    movel([0.119782, -1.382241, -2.558201, -0.771947, 1.570796, 1.690578],accel_mss,speed_ms,0,blend_radius_m)
    speed_ms = 1.000
    movel([0.119782, -1.357452, -2.545969, -0.808968, 1.570796, 1.690578],accel_mss,speed_ms,0,blend_radius_m)
    movel([0.118569, -1.359477, -2.544576, -0.808336, 1.570796, 1.689365],accel_mss,speed_ms,0,blend_radius_m)
    movel([0.118569, -1.384229, -2.556783, -0.771377, 1.570796, 1.689365],accel_mss,speed_ms,0,blend_radius_m)
    speed_ms = 0.003
    movel([0.118569, -1.393867, -2.561225, -0.757297, 1.570796, 1.689365],accel_mss,speed_ms,0,blend_radius_m)
    speed_ms = 0.007
    movel([0.118728, -1.394054, -2.561089, -0.757246, 1.570796, 1.689524],accel_mss,speed_ms,0,blend_radius_m)
    movel([0.118593, -1.394865, -2.560501, -0.757024, 1.570796, 1.689390],accel_mss,speed_ms,0,blend_radius_m)
    movel([0.118424, -1.395809, -2.559814, -0.756766, 1.570796, 1.689220],accel_mss,speed_ms,0,blend_radius_m)
    movel([0.118206, -1.396901, -2.559018, -0.756470, 1.570796, 1.689002],accel_mss,speed_ms,0,blend_radius_m)
    movel([0.117896, -1.398373, -2.557942, -0.756074, 1.570796, 1.688693],accel_mss,speed_ms,0,blend_radius_m)
    movel([0.117699, -1.399201, -2.557336, -0.755852, 1.570796, 1.688495],accel_mss,speed_ms,0,blend_radius_m)
    movel([0.117545, -1.399729, -2.556948, -0.755712, 1.570796, 1.688341],accel_mss,speed_ms,0,blend_radius_m)
    movel([0.117303, -1.400036, -2.556723, -0.755630, 1.570796, 1.688099],accel_mss,speed_ms,0,blend_radius_m)
    movel([0.117055, -1.400079, -2.556692, -0.755619, 1.570796, 1.687851],accel_mss,speed_ms,0,blend_radius_m)
    movel([0.117023, -1.399429, -2.557168, -0.755792, 1.570796, 1.687819],accel_mss,speed_ms,0,blend_radius_m)
    movel([0.117111, -1.398603, -2.557774, -0.756012, 1.570796, 1.687907],accel_mss,speed_ms,0,blend_radius_m)
    movel([0.117305, -1.397157, -2.558831, -0.756401, 1.570796, 1.688101],accel_mss,speed_ms,0,blend_radius_m)
    movel([0.117464, -1.396051, -2.559637, -0.756700, 1.570796, 1.688261],accel_mss,speed_ms,0,blend_radius_m)
    movel([0.117616, -1.395092, -2.560336, -0.756962, 1.570796, 1.688412],accel_mss,speed_ms,0,blend_radius_m)
    movel([0.117758, -1.394259, -2.560940, -0.757189, 1.570796, 1.688554],accel_mss,speed_ms,0,blend_radius_m)
    movel([0.117985, -1.394001, -2.561128, -0.757260, 1.570796, 1.688781],accel_mss,speed_ms,0,blend_radius_m)
    movel([0.118280, -1.393900, -2.561201, -0.757288, 1.570796, 1.689077],accel_mss,speed_ms,0,blend_radius_m)
    movel([0.118569, -1.393867, -2.561225, -0.757297, 1.570796, 1.689365],accel_mss,speed_ms,0,blend_radius_m)
    speed_ms = 0.003
    movel([0.118569, -1.397123, -2.562689, -0.752577, 1.570796, 1.689365],accel_mss,speed_ms,0,blend_radius_m)
    speed_ms = 0.007
    movel([0.118728, -1.397310, -2.562553, -0.752526, 1.570796, 1.689524],accel_mss,speed_ms,0,blend_radius_m)
    movel([0.118593, -1.398118, -2.561963, -0.752308, 1.570796, 1.689390],accel_mss,speed_ms,0,blend_radius_m)
    movel([0.118424, -1.399059, -2.561275, -0.752055, 1.570796, 1.689220],accel_mss,speed_ms,0,blend_radius_m)
    movel([0.118206, -1.400148, -2.560477, -0.751764, 1.570796, 1.689002],accel_mss,speed_ms,0,blend_radius_m)
    movel([0.117896, -1.401617, -2.559399, -0.751374, 1.570796, 1.688693],accel_mss,speed_ms,0,blend_radius_m)
    movel([0.117699, -1.402442, -2.558791, -0.751156, 1.570796, 1.688495],accel_mss,speed_ms,0,blend_radius_m)
    movel([0.117545, -1.402968, -2.558403, -0.751018, 1.570796, 1.688341],accel_mss,speed_ms,0,blend_radius_m)
    movel([0.117303, -1.403274, -2.558177, -0.750937, 1.570796, 1.688099],accel_mss,speed_ms,0,blend_radius_m)
    movel([0.117055, -1.403317, -2.558145, -0.750926, 1.570796, 1.687851],accel_mss,speed_ms,0,blend_radius_m)
    movel([0.117023, -1.402670, -2.558623, -0.751096, 1.570796, 1.687819],accel_mss,speed_ms,0,blend_radius_m)
    movel([0.117111, -1.401846, -2.559230, -0.751313, 1.570796, 1.687907],accel_mss,speed_ms,0,blend_radius_m)
    movel([0.117305, -1.400404, -2.560290, -0.751696, 1.570796, 1.688101],accel_mss,speed_ms,0,blend_radius_m)
    movel([0.117464, -1.399301, -2.561098, -0.751990, 1.570796, 1.688261],accel_mss,speed_ms,0,blend_radius_m)
    movel([0.117616, -1.398344, -2.561798, -0.752247, 1.570796, 1.688412],accel_mss,speed_ms,0,blend_radius_m)
    movel([0.117758, -1.397514, -2.562404, -0.752471, 1.570796, 1.688554],accel_mss,speed_ms,0,blend_radius_m)
    movel([0.117985, -1.397256, -2.562592, -0.752541, 1.570796, 1.688781],accel_mss,speed_ms,0,blend_radius_m)
    movel([0.118280, -1.397156, -2.562665, -0.752568, 1.570796, 1.689077],accel_mss,speed_ms,0,blend_radius_m)
    movel([0.118569, -1.397123, -2.562689, -0.752577, 1.570796, 1.689365],accel_mss,speed_ms,0,blend_radius_m)
    speed_ms = 0.003
    movel([0.118569, -1.384229, -2.556783, -0.771377, 1.570796, 1.689365],accel_mss,speed_ms,0,blend_radius_m)
    speed_ms = 1.000
    movel([0.118569, -1.359477, -2.544576, -0.808336, 1.570796, 1.689365],accel_mss,speed_ms,0,blend_radius_m)
    movel([0.118605, -1.358852, -2.545007, -0.808530, 1.570796, 1.689401],accel_mss,speed_ms,0,blend_radius_m)
    movel([0.118605, -1.383615, -2.557221, -0.771552, 1.570796, 1.689401],accel_mss,speed_ms,0,blend_radius_m)
    speed_ms = 0.003
    movel([0.118605, -1.393258, -2.561667, -0.757465, 1.570796, 1.689401],accel_mss,speed_ms,0,blend_radius_m)
    speed_ms = 0.007
    movel([0.118234, -1.393393, -2.561569, -0.757427, 1.570796, 1.689030],accel_mss,speed_ms,0,blend_radius_m)
    movel([0.117908, -1.393450, -2.561527, -0.757412, 1.570796, 1.688705],accel_mss,speed_ms,0,blend_radius_m)
    movel([0.117689, -1.393424, -2.561546, -0.757419, 1.570796, 1.688485],accel_mss,speed_ms,0,blend_radius_m)
    movel([0.117549, -1.393131, -2.561759, -0.757500, 1.570796, 1.688345],accel_mss,speed_ms,0,blend_radius_m)
    movel([0.117522, -1.392806, -2.561994, -0.757589, 1.570796, 1.688318],accel_mss,speed_ms,0,blend_radius_m)
    movel([0.117346, -1.392422, -2.562271, -0.757695, 1.570796, 1.688142],accel_mss,speed_ms,0,blend_radius_m)
    movel([0.117088, -1.392080, -2.562518, -0.757790, 1.570796, 1.687885],accel_mss,speed_ms,0,blend_radius_m)
    movel([0.116802, -1.391882, -2.562661, -0.757845, 1.570796, 1.687598],accel_mss,speed_ms,0,blend_radius_m)
    movel([0.116439, -1.391787, -2.562731, -0.757872, 1.570796, 1.687236],accel_mss,speed_ms,0,blend_radius_m)
    movel([0.116040, -1.391804, -2.562718, -0.757867, 1.570796, 1.686837],accel_mss,speed_ms,0,blend_radius_m)
    movel([0.115619, -1.391935, -2.562624, -0.757831, 1.570796, 1.686415],accel_mss,speed_ms,0,blend_radius_m)
    movel([0.115183, -1.392176, -2.562449, -0.757764, 1.570796, 1.685979],accel_mss,speed_ms,0,blend_radius_m)
    movel([0.114712, -1.392597, -2.562145, -0.757647, 1.570796, 1.685508],accel_mss,speed_ms,0,blend_radius_m)
    movel([0.114471, -1.393051, -2.561816, -0.757522, 1.570796, 1.685267],accel_mss,speed_ms,0,blend_radius_m)
    movel([0.114501, -1.393491, -2.561498, -0.757401, 1.570796, 1.685297],accel_mss,speed_ms,0,blend_radius_m)
    movel([0.114790, -1.393868, -2.561224, -0.757297, 1.570796, 1.685586],accel_mss,speed_ms,0,blend_radius_m)
    movel([0.115093, -1.394046, -2.561095, -0.757248, 1.570796, 1.685889],accel_mss,speed_ms,0,blend_radius_m)
    movel([0.115465, -1.394151, -2.561019, -0.757219, 1.570796, 1.686262],accel_mss,speed_ms,0,blend_radius_m)
    movel([0.115948, -1.394188, -2.560992, -0.757209, 1.570796, 1.686745],accel_mss,speed_ms,0,blend_radius_m)
    movel([0.116596, -1.394166, -2.561008, -0.757215, 1.570796, 1.687392],accel_mss,speed_ms,0,blend_radius_m)
    movel([0.116840, -1.394198, -2.560985, -0.757206, 1.570796, 1.687637],accel_mss,speed_ms,0,blend_radius_m)
    movel([0.117037, -1.394702, -2.560619, -0.757068, 1.570796, 1.687833],accel_mss,speed_ms,0,blend_radius_m)
    movel([0.116741, -1.397152, -2.558834, -0.756402, 1.570796, 1.687538],accel_mss,speed_ms,0,blend_radius_m)
    movel([0.116430, -1.399585, -2.557054, -0.755750, 1.570796, 1.687226],accel_mss,speed_ms,0,blend_radius_m)
    movel([0.116267, -1.400079, -2.556692, -0.755619, 1.570796, 1.687063],accel_mss,speed_ms,0,blend_radius_m)
    movel([0.116071, -1.400343, -2.556497, -0.755549, 1.570796, 1.686867],accel_mss,speed_ms,0,blend_radius_m)
    movel([0.115806, -1.400476, -2.556399, -0.755513, 1.570796, 1.686603],accel_mss,speed_ms,0,blend_radius_m)
    movel([0.115532, -1.400483, -2.556394, -0.755511, 1.570796, 1.686329],accel_mss,speed_ms,0,blend_radius_m)
    movel([0.115371, -1.400354, -2.556490, -0.755546, 1.570796, 1.686167],accel_mss,speed_ms,0,blend_radius_m)
    movel([0.115306, -1.400032, -2.556726, -0.755631, 1.570796, 1.686102],accel_mss,speed_ms,0,blend_radius_m)
    movel([0.115324, -1.399384, -2.557202, -0.755804, 1.570796, 1.686120],accel_mss,speed_ms,0,blend_radius_m)
    movel([0.115335, -1.399019, -2.557469, -0.755901, 1.570796, 1.686131],accel_mss,speed_ms,0,blend_radius_m)
    movel([0.115328, -1.398702, -2.557701, -0.755986, 1.570796, 1.686124],accel_mss,speed_ms,0,blend_radius_m)
    movel([0.115303, -1.398449, -2.557887, -0.756054, 1.570796, 1.686099],accel_mss,speed_ms,0,blend_radius_m)
    movel([0.114943, -1.398374, -2.557941, -0.756074, 1.570796, 1.685739],accel_mss,speed_ms,0,blend_radius_m)
    movel([0.114662, -1.398389, -2.557930, -0.756070, 1.570796, 1.685459],accel_mss,speed_ms,0,blend_radius_m)
    movel([0.114357, -1.398417, -2.557910, -0.756062, 1.570796, 1.685153],accel_mss,speed_ms,0,blend_radius_m)
    movel([0.112719, -1.398331, -2.557973, -0.756085, 1.570796, 1.683515],accel_mss,speed_ms,0,blend_radius_m)
    movel([0.111315, -1.397718, -2.558421, -0.756250, 1.570796, 1.682112],accel_mss,speed_ms,0,blend_radius_m)
    movel([0.110329, -1.396670, -2.559187, -0.756533, 1.570796, 1.681125],accel_mss,speed_ms,0,blend_radius_m)
    movel([0.109898, -1.395312, -2.560175, -0.756901, 1.570796, 1.680695],accel_mss,speed_ms,0,blend_radius_m)
    movel([0.110008, -1.393931, -2.561179, -0.757279, 1.570796, 1.680804],accel_mss,speed_ms,0,blend_radius_m)
    movel([0.110561, -1.392374, -2.562306, -0.757709, 1.570796, 1.681357],accel_mss,speed_ms,0,blend_radius_m)
    movel([0.111504, -1.390778, -2.563459, -0.758153, 1.570796, 1.682300],accel_mss,speed_ms,0,blend_radius_m)
    movel([0.112755, -1.389292, -2.564528, -0.758569, 1.570796, 1.683551],accel_mss,speed_ms,0,blend_radius_m)
    movel([0.113901, -1.388249, -2.565277, -0.758863, 1.570796, 1.684697],accel_mss,speed_ms,0,blend_radius_m)
    movel([0.115113, -1.387370, -2.565906, -0.759112, 1.570796, 1.685909],accel_mss,speed_ms,0,blend_radius_m)
    movel([0.116414, -1.386641, -2.566428, -0.759320, 1.570796, 1.687210],accel_mss,speed_ms,0,blend_radius_m)
    movel([0.117832, -1.386048, -2.566851, -0.759489, 1.570796, 1.688629],accel_mss,speed_ms,0,blend_radius_m)
    movel([0.119207, -1.385643, -2.567141, -0.759605, 1.570796, 1.690004],accel_mss,speed_ms,0,blend_radius_m)
    movel([0.120533, -1.385423, -2.567298, -0.759669, 1.570796, 1.691329],accel_mss,speed_ms,0,blend_radius_m)
    movel([0.121802, -1.385387, -2.567323, -0.759679, 1.570796, 1.692598],accel_mss,speed_ms,0,blend_radius_m)
    movel([0.123004, -1.385538, -2.567216, -0.759636, 1.570796, 1.693800],accel_mss,speed_ms,0,blend_radius_m)
    movel([0.124432, -1.386000, -2.566886, -0.759503, 1.570796, 1.695228],accel_mss,speed_ms,0,blend_radius_m)
    movel([0.125530, -1.386717, -2.566374, -0.759299, 1.570796, 1.696327],accel_mss,speed_ms,0,blend_radius_m)
    movel([0.126289, -1.387678, -2.565686, -0.759025, 1.570796, 1.697085],accel_mss,speed_ms,0,blend_radius_m)
    movel([0.126698, -1.388871, -2.564830, -0.758688, 1.570796, 1.697494],accel_mss,speed_ms,0,blend_radius_m)
    movel([0.126745, -1.389618, -2.564293, -0.758477, 1.570796, 1.697542],accel_mss,speed_ms,0,blend_radius_m)
    movel([0.126649, -1.390509, -2.563652, -0.758228, 1.570796, 1.697445],accel_mss,speed_ms,0,blend_radius_m)
    movel([0.126428, -1.391420, -2.562996, -0.757974, 1.570796, 1.697225],accel_mss,speed_ms,0,blend_radius_m)
    movel([0.126106, -1.392220, -2.562417, -0.757751, 1.570796, 1.696902],accel_mss,speed_ms,0,blend_radius_m)
    movel([0.125118, -1.393737, -2.561319, -0.757333, 1.570796, 1.695914],accel_mss,speed_ms,0,blend_radius_m)
    movel([0.123745, -1.395105, -2.560326, -0.756958, 1.570796, 1.694541],accel_mss,speed_ms,0,blend_radius_m)
    movel([0.122153, -1.396174, -2.559548, -0.756667, 1.570796, 1.692950],accel_mss,speed_ms,0,blend_radius_m)
    movel([0.120525, -1.396815, -2.559081, -0.756494, 1.570796, 1.691322],accel_mss,speed_ms,0,blend_radius_m)
    movel([0.120253, -1.396893, -2.559024, -0.756473, 1.570796, 1.691049],accel_mss,speed_ms,0,blend_radius_m)
    movel([0.119842, -1.397065, -2.558898, -0.756426, 1.570796, 1.690638],accel_mss,speed_ms,0,blend_radius_m)
    movel([0.119569, -1.397624, -2.558489, -0.756275, 1.570796, 1.690365],accel_mss,speed_ms,0,blend_radius_m)
    movel([0.119430, -1.398068, -2.558166, -0.756156, 1.570796, 1.690226],accel_mss,speed_ms,0,blend_radius_m)
    movel([0.119286, -1.398565, -2.557802, -0.756023, 1.570796, 1.690082],accel_mss,speed_ms,0,blend_radius_m)
    movel([0.119073, -1.399308, -2.557257, -0.755824, 1.570796, 1.689869],accel_mss,speed_ms,0,blend_radius_m)
    movel([0.118949, -1.399640, -2.557014, -0.755735, 1.570796, 1.689746],accel_mss,speed_ms,0,blend_radius_m)
    movel([0.118677, -1.399926, -2.556804, -0.755659, 1.570796, 1.689474],accel_mss,speed_ms,0,blend_radius_m)
    movel([0.118374, -1.399909, -2.556816, -0.755664, 1.570796, 1.689170],accel_mss,speed_ms,0,blend_radius_m)
    movel([0.118256, -1.399637, -2.557016, -0.755736, 1.570796, 1.689052],accel_mss,speed_ms,0,blend_radius_m)
    movel([0.118338, -1.398896, -2.557559, -0.755934, 1.570796, 1.689135],accel_mss,speed_ms,0,blend_radius_m)
    movel([0.118759, -1.396778, -2.559108, -0.756504, 1.570796, 1.689555],accel_mss,speed_ms,0,blend_radius_m)
    movel([0.119135, -1.394964, -2.560428, -0.756997, 1.570796, 1.689932],accel_mss,speed_ms,0,blend_radius_m)
    movel([0.119322, -1.394196, -2.560986, -0.757207, 1.570796, 1.690118],accel_mss,speed_ms,0,blend_radius_m)
    movel([0.119471, -1.393764, -2.561299, -0.757325, 1.570796, 1.690267],accel_mss,speed_ms,0,blend_radius_m)
    movel([0.119650, -1.393519, -2.561478, -0.757393, 1.570796, 1.690446],accel_mss,speed_ms,0,blend_radius_m)
    movel([0.119894, -1.393328, -2.561616, -0.757445, 1.570796, 1.690690],accel_mss,speed_ms,0,blend_radius_m)
    movel([0.120184, -1.393181, -2.561722, -0.757486, 1.570796, 1.690980],accel_mss,speed_ms,0,blend_radius_m)
    movel([0.120541, -1.392912, -2.561917, -0.757560, 1.570796, 1.691338],accel_mss,speed_ms,0,blend_radius_m)
    movel([0.121356, -1.391952, -2.562611, -0.757826, 1.570796, 1.692152],accel_mss,speed_ms,0,blend_radius_m)
    movel([0.121511, -1.391218, -2.563141, -0.758030, 1.570796, 1.692307],accel_mss,speed_ms,0,blend_radius_m)
    movel([0.121159, -1.390779, -2.563458, -0.758152, 1.570796, 1.691955],accel_mss,speed_ms,0,blend_radius_m)
    movel([0.120423, -1.390764, -2.563469, -0.758157, 1.570796, 1.691219],accel_mss,speed_ms,0,blend_radius_m)
    movel([0.119974, -1.390949, -2.563335, -0.758105, 1.570796, 1.690770],accel_mss,speed_ms,0,blend_radius_m)
    movel([0.119626, -1.391236, -2.563128, -0.758025, 1.570796, 1.690422],accel_mss,speed_ms,0,blend_radius_m)
    movel([0.119362, -1.391651, -2.562829, -0.757909, 1.570796, 1.690158],accel_mss,speed_ms,0,blend_radius_m)
    movel([0.119164, -1.392229, -2.562411, -0.757749, 1.570796, 1.689960],accel_mss,speed_ms,0,blend_radius_m)
    movel([0.118997, -1.392786, -2.562008, -0.757595, 1.570796, 1.689793],accel_mss,speed_ms,0,blend_radius_m)
    movel([0.118834, -1.393077, -2.561797, -0.757514, 1.570796, 1.689630],accel_mss,speed_ms,0,blend_radius_m)
    movel([0.118605, -1.393258, -2.561667, -0.757465, 1.570796, 1.689401],accel_mss,speed_ms,0,blend_radius_m)
    speed_ms = 0.003
    movel([0.118605, -1.396515, -2.563132, -0.752742, 1.570796, 1.689401],accel_mss,speed_ms,0,blend_radius_m)
    speed_ms = 0.007
    movel([0.118234, -1.396650, -2.563034, -0.752705, 1.570796, 1.689030],accel_mss,speed_ms,0,blend_radius_m)
    movel([0.117908, -1.396707, -2.562992, -0.752690, 1.570796, 1.688705],accel_mss,speed_ms,0,blend_radius_m)
    movel([0.117689, -1.396681, -2.563011, -0.752697, 1.570796, 1.688485],accel_mss,speed_ms,0,blend_radius_m)
    movel([0.117549, -1.396389, -2.563224, -0.752776, 1.570796, 1.688345],accel_mss,speed_ms,0,blend_radius_m)
    movel([0.117522, -1.396065, -2.563460, -0.752865, 1.570796, 1.688318],accel_mss,speed_ms,0,blend_radius_m)
    movel([0.117346, -1.395682, -2.563738, -0.752969, 1.570796, 1.688142],accel_mss,speed_ms,0,blend_radius_m)
    movel([0.117088, -1.395341, -2.563985, -0.753062, 1.570796, 1.687885],accel_mss,speed_ms,0,blend_radius_m)
    movel([0.116802, -1.395144, -2.564129, -0.753116, 1.570796, 1.687598],accel_mss,speed_ms,0,blend_radius_m)
    movel([0.116439, -1.395048, -2.564198, -0.753143, 1.570796, 1.687236],accel_mss,speed_ms,0,blend_radius_m)
    movel([0.116040, -1.395066, -2.564185, -0.753138, 1.570796, 1.686837],accel_mss,speed_ms,0,blend_radius_m)
    movel([0.115619, -1.395196, -2.564091, -0.753102, 1.570796, 1.686415],accel_mss,speed_ms,0,blend_radius_m)
    movel([0.115183, -1.395437, -2.563916, -0.753036, 1.570796, 1.685979],accel_mss,speed_ms,0,blend_radius_m)
    movel([0.114712, -1.395856, -2.563611, -0.752922, 1.570796, 1.685508],accel_mss,speed_ms,0,blend_radius_m)
    movel([0.114471, -1.396309, -2.563281, -0.752798, 1.570796, 1.685267],accel_mss,speed_ms,0,blend_radius_m)
    movel([0.114501, -1.396748, -2.562962, -0.752679, 1.570796, 1.685297],accel_mss,speed_ms,0,blend_radius_m)
    movel([0.114790, -1.397124, -2.562688, -0.752577, 1.570796, 1.685586],accel_mss,speed_ms,0,blend_radius_m)
    movel([0.115093, -1.397302, -2.562559, -0.752529, 1.570796, 1.685889],accel_mss,speed_ms,0,blend_radius_m)
    movel([0.115465, -1.397406, -2.562482, -0.752500, 1.570796, 1.686262],accel_mss,speed_ms,0,blend_radius_m)
    movel([0.115948, -1.397443, -2.562455, -0.752490, 1.570796, 1.686745],accel_mss,speed_ms,0,blend_radius_m)
    movel([0.116596, -1.397422, -2.562471, -0.752496, 1.570796, 1.687392],accel_mss,speed_ms,0,blend_radius_m)
    movel([0.116840, -1.397453, -2.562448, -0.752488, 1.570796, 1.687637],accel_mss,speed_ms,0,blend_radius_m)
    movel([0.117037, -1.397956, -2.562081, -0.752352, 1.570796, 1.687833],accel_mss,speed_ms,0,blend_radius_m)
    movel([0.116741, -1.400399, -2.560293, -0.751697, 1.570796, 1.687538],accel_mss,speed_ms,0,blend_radius_m)
    movel([0.116430, -1.402825, -2.558508, -0.751055, 1.570796, 1.687226],accel_mss,speed_ms,0,blend_radius_m)
    movel([0.116267, -1.403317, -2.558146, -0.750926, 1.570796, 1.687063],accel_mss,speed_ms,0,blend_radius_m)
    movel([0.116071, -1.403581, -2.557951, -0.750857, 1.570796, 1.686867],accel_mss,speed_ms,0,blend_radius_m)
    movel([0.115806, -1.403714, -2.557853, -0.750822, 1.570796, 1.686603],accel_mss,speed_ms,0,blend_radius_m)
    movel([0.115532, -1.403721, -2.557848, -0.750821, 1.570796, 1.686329],accel_mss,speed_ms,0,blend_radius_m)
    movel([0.115371, -1.403591, -2.557943, -0.750854, 1.570796, 1.686167],accel_mss,speed_ms,0,blend_radius_m)
    movel([0.115306, -1.403270, -2.558180, -0.750938, 1.570796, 1.686102],accel_mss,speed_ms,0,blend_radius_m)
    movel([0.115324, -1.402624, -2.558657, -0.751108, 1.570796, 1.686120],accel_mss,speed_ms,0,blend_radius_m)
    movel([0.115335, -1.402261, -2.558925, -0.751204, 1.570796, 1.686131],accel_mss,speed_ms,0,blend_radius_m)
    movel([0.115328, -1.401944, -2.559157, -0.751287, 1.570796, 1.686124],accel_mss,speed_ms,0,blend_radius_m)
    movel([0.115303, -1.401692, -2.559343, -0.751354, 1.570796, 1.686099],accel_mss,speed_ms,0,blend_radius_m)
    movel([0.114943, -1.401617, -2.559398, -0.751374, 1.570796, 1.685739],accel_mss,speed_ms,0,blend_radius_m)
    movel([0.114662, -1.401633, -2.559387, -0.751370, 1.570796, 1.685459],accel_mss,speed_ms,0,blend_radius_m)
    movel([0.114357, -1.401660, -2.559366, -0.751362, 1.570796, 1.685153],accel_mss,speed_ms,0,blend_radius_m)
    movel([0.112719, -1.401575, -2.559429, -0.751385, 1.570796, 1.683515],accel_mss,speed_ms,0,blend_radius_m)
    movel([0.111315, -1.400963, -2.559879, -0.751547, 1.570796, 1.682112],accel_mss,speed_ms,0,blend_radius_m)
    movel([0.110329, -1.399918, -2.560646, -0.751825, 1.570796, 1.681125],accel_mss,speed_ms,0,blend_radius_m)
    movel([0.109898, -1.398564, -2.561637, -0.752188, 1.570796, 1.680695],accel_mss,speed_ms,0,blend_radius_m)
    movel([0.110008, -1.397187, -2.562642, -0.752560, 1.570796, 1.680804],accel_mss,speed_ms,0,blend_radius_m)
    movel([0.110561, -1.395634, -2.563773, -0.752982, 1.570796, 1.681357],accel_mss,speed_ms,0,blend_radius_m)
    movel([0.111504, -1.394042, -2.564928, -0.753419, 1.570796, 1.682300],accel_mss,speed_ms,0,blend_radius_m)
    movel([0.112755, -1.392561, -2.565999, -0.753829, 1.570796, 1.683551],accel_mss,speed_ms,0,blend_radius_m)
    movel([0.113901, -1.391520, -2.566750, -0.754119, 1.570796, 1.684697],accel_mss,speed_ms,0,blend_radius_m)
    movel([0.115113, -1.390644, -2.567381, -0.754364, 1.570796, 1.685909],accel_mss,speed_ms,0,blend_radius_m)
    movel([0.116414, -1.389917, -2.567904, -0.754568, 1.570796, 1.687210],accel_mss,speed_ms,0,blend_radius_m)
    movel([0.117832, -1.389326, -2.568328, -0.754735, 1.570796, 1.688629],accel_mss,speed_ms,0,blend_radius_m)
    movel([0.119207, -1.388922, -2.568618, -0.754849, 1.570796, 1.690004],accel_mss,speed_ms,0,blend_radius_m)
    movel([0.120533, -1.388702, -2.568775, -0.754912, 1.570796, 1.691329],accel_mss,speed_ms,0,blend_radius_m)
    movel([0.121802, -1.388667, -2.568801, -0.754922, 1.570796, 1.692598],accel_mss,speed_ms,0,blend_radius_m)
    movel([0.123004, -1.388816, -2.568693, -0.754879, 1.570796, 1.693800],accel_mss,speed_ms,0,blend_radius_m)
    movel([0.124432, -1.389277, -2.568363, -0.754749, 1.570796, 1.695228],accel_mss,speed_ms,0,blend_radius_m)
    movel([0.125530, -1.389992, -2.567850, -0.754547, 1.570796, 1.696327],accel_mss,speed_ms,0,blend_radius_m)
    movel([0.126289, -1.390951, -2.567160, -0.754278, 1.570796, 1.697085],accel_mss,speed_ms,0,blend_radius_m)
    movel([0.126698, -1.392141, -2.566302, -0.753946, 1.570796, 1.697494],accel_mss,speed_ms,0,blend_radius_m)
    movel([0.126745, -1.392886, -2.565764, -0.753739, 1.570796, 1.697542],accel_mss,speed_ms,0,blend_radius_m)
    movel([0.126649, -1.393774, -2.565122, -0.753493, 1.570796, 1.697445],accel_mss,speed_ms,0,blend_radius_m)
    movel([0.126428, -1.394682, -2.564464, -0.753243, 1.570796, 1.697225],accel_mss,speed_ms,0,blend_radius_m)
    movel([0.126106, -1.395481, -2.563884, -0.753024, 1.570796, 1.696902],accel_mss,speed_ms,0,blend_radius_m)
    movel([0.125118, -1.396993, -2.562784, -0.752612, 1.570796, 1.695914],accel_mss,speed_ms,0,blend_radius_m)
    movel([0.123745, -1.398357, -2.561788, -0.752244, 1.570796, 1.694541],accel_mss,speed_ms,0,blend_radius_m)
    movel([0.122153, -1.399423, -2.561008, -0.751957, 1.570796, 1.692950],accel_mss,speed_ms,0,blend_radius_m)
    movel([0.120525, -1.400063, -2.560540, -0.751787, 1.570796, 1.691322],accel_mss,speed_ms,0,blend_radius_m)
    movel([0.120253, -1.400140, -2.560483, -0.751766, 1.570796, 1.691049],accel_mss,speed_ms,0,blend_radius_m)
    movel([0.119842, -1.400312, -2.560357, -0.751720, 1.570796, 1.690638],accel_mss,speed_ms,0,blend_radius_m)
    movel([0.119569, -1.400870, -2.559947, -0.751572, 1.570796, 1.690365],accel_mss,speed_ms,0,blend_radius_m)
    movel([0.119430, -1.401312, -2.559623, -0.751455, 1.570796, 1.690226],accel_mss,speed_ms,0,blend_radius_m)
    movel([0.119286, -1.401808, -2.559258, -0.751323, 1.570796, 1.690082],accel_mss,speed_ms,0,blend_radius_m)
    movel([0.119073, -1.402549, -2.558712, -0.751128, 1.570796, 1.689869],accel_mss,speed_ms,0,blend_radius_m)
    movel([0.118949, -1.402880, -2.558468, -0.751041, 1.570796, 1.689746],accel_mss,speed_ms,0,blend_radius_m)
    movel([0.118677, -1.403165, -2.558258, -0.750966, 1.570796, 1.689474],accel_mss,speed_ms,0,blend_radius_m)
    movel([0.118374, -1.403148, -2.558270, -0.750970, 1.570796, 1.689170],accel_mss,speed_ms,0,blend_radius_m)
    movel([0.118256, -1.402877, -2.558470, -0.751042, 1.570796, 1.689052],accel_mss,speed_ms,0,blend_radius_m)
    movel([0.118338, -1.402138, -2.559015, -0.751236, 1.570796, 1.689135],accel_mss,speed_ms,0,blend_radius_m)
    movel([0.118759, -1.400026, -2.560567, -0.751796, 1.570796, 1.689555],accel_mss,speed_ms,0,blend_radius_m)
    movel([0.119135, -1.398217, -2.561891, -0.752281, 1.570796, 1.689932],accel_mss,speed_ms,0,blend_radius_m)
    movel([0.119322, -1.397451, -2.562450, -0.752488, 1.570796, 1.690118],accel_mss,speed_ms,0,blend_radius_m)
    movel([0.119471, -1.397021, -2.562764, -0.752605, 1.570796, 1.690267],accel_mss,speed_ms,0,blend_radius_m)
    movel([0.119650, -1.396776, -2.562942, -0.752671, 1.570796, 1.690446],accel_mss,speed_ms,0,blend_radius_m)
    movel([0.119894, -1.396586, -2.563080, -0.752723, 1.570796, 1.690690],accel_mss,speed_ms,0,blend_radius_m)
    movel([0.120184, -1.396439, -2.563187, -0.752763, 1.570796, 1.690980],accel_mss,speed_ms,0,blend_radius_m)
    movel([0.120541, -1.396171, -2.563382, -0.752836, 1.570796, 1.691338],accel_mss,speed_ms,0,blend_radius_m)
    movel([0.121356, -1.395214, -2.564078, -0.753097, 1.570796, 1.692152],accel_mss,speed_ms,0,blend_radius_m)
    movel([0.121511, -1.394481, -2.564609, -0.753298, 1.570796, 1.692307],accel_mss,speed_ms,0,blend_radius_m)
    movel([0.121159, -1.394043, -2.564927, -0.753419, 1.570796, 1.691955],accel_mss,speed_ms,0,blend_radius_m)
    movel([0.120423, -1.394028, -2.564938, -0.753423, 1.570796, 1.691219],accel_mss,speed_ms,0,blend_radius_m)
    movel([0.119974, -1.394213, -2.564804, -0.753372, 1.570796, 1.690770],accel_mss,speed_ms,0,blend_radius_m)
    movel([0.119626, -1.394499, -2.564597, -0.753293, 1.570796, 1.690422],accel_mss,speed_ms,0,blend_radius_m)
    movel([0.119362, -1.394913, -2.564296, -0.753180, 1.570796, 1.690158],accel_mss,speed_ms,0,blend_radius_m)
    movel([0.119164, -1.395489, -2.563878, -0.753022, 1.570796, 1.689960],accel_mss,speed_ms,0,blend_radius_m)
    movel([0.118997, -1.396045, -2.563474, -0.752870, 1.570796, 1.689793],accel_mss,speed_ms,0,blend_radius_m)
    movel([0.118834, -1.396335, -2.563263, -0.752791, 1.570796, 1.689630],accel_mss,speed_ms,0,blend_radius_m)
    movel([0.118605, -1.396515, -2.563132, -0.752742, 1.570796, 1.689401],accel_mss,speed_ms,0,blend_radius_m)
    speed_ms = 0.003
    movel([0.118605, -1.383615, -2.557221, -0.771552, 1.570796, 1.689401],accel_mss,speed_ms,0,blend_radius_m)
    speed_ms = 1.000
    movel([0.118605, -1.358852, -2.545007, -0.808530, 1.570796, 1.689401],accel_mss,speed_ms,0,blend_radius_m)
    movel([0.116923, -1.366587, -2.539643, -0.806159, 1.570796, 1.687720],accel_mss,speed_ms,0,blend_radius_m)
    movel([0.116923, -1.391208, -2.551760, -0.769421, 1.570796, 1.687720],accel_mss,speed_ms,0,blend_radius_m)
    speed_ms = 0.003
    movel([0.116923, -1.400790, -2.556169, -0.755430, 1.570796, 1.687720],accel_mss,speed_ms,0,blend_radius_m)
    speed_ms = 0.007
    movel([0.118450, -1.400541, -2.556352, -0.755496, 1.570796, 1.689246],accel_mss,speed_ms,0,blend_radius_m)
    movel([0.119164, -1.400486, -2.556392, -0.755511, 1.570796, 1.689961],accel_mss,speed_ms,0,blend_radius_m)
    movel([0.119522, -1.400571, -2.556330, -0.755488, 1.570796, 1.690318],accel_mss,speed_ms,0,blend_radius_m)
    movel([0.119673, -1.400804, -2.556159, -0.755426, 1.570796, 1.690469],accel_mss,speed_ms,0,blend_radius_m)
    movel([0.119491, -1.401099, -2.555942, -0.755349, 1.570796, 1.690287],accel_mss,speed_ms,0,blend_radius_m)
    movel([0.119212, -1.401506, -2.555642, -0.755241, 1.570796, 1.690008],accel_mss,speed_ms,0,blend_radius_m)
    movel([0.119126, -1.401821, -2.555410, -0.755158, 1.570796, 1.689922],accel_mss,speed_ms,0,blend_radius_m)
    movel([0.119166, -1.402025, -2.555260, -0.755105, 1.570796, 1.689962],accel_mss,speed_ms,0,blend_radius_m)
    movel([0.119206, -1.402226, -2.555111, -0.755052, 1.570796, 1.690002],accel_mss,speed_ms,0,blend_radius_m)
    movel([0.119129, -1.402510, -2.554902, -0.754977, 1.570796, 1.689926],accel_mss,speed_ms,0,blend_radius_m)
    movel([0.118545, -1.403144, -2.554433, -0.754811, 1.570796, 1.689342],accel_mss,speed_ms,0,blend_radius_m)
    movel([0.118026, -1.403479, -2.554186, -0.754724, 1.570796, 1.688823],accel_mss,speed_ms,0,blend_radius_m)
    movel([0.117329, -1.403764, -2.553976, -0.754650, 1.570796, 1.688126],accel_mss,speed_ms,0,blend_radius_m)
    movel([0.116307, -1.404052, -2.553762, -0.754575, 1.570796, 1.687103],accel_mss,speed_ms,0,blend_radius_m)
    movel([0.115098, -1.404316, -2.553567, -0.754506, 1.570796, 1.685894],accel_mss,speed_ms,0,blend_radius_m)
    movel([0.114445, -1.404324, -2.553560, -0.754504, 1.570796, 1.685242],accel_mss,speed_ms,0,blend_radius_m)
    movel([0.114245, -1.404102, -2.553725, -0.754562, 1.570796, 1.685042],accel_mss,speed_ms,0,blend_radius_m)
    movel([0.114389, -1.403691, -2.554029, -0.754669, 1.570796, 1.685185],accel_mss,speed_ms,0,blend_radius_m)
    movel([0.114487, -1.403461, -2.554199, -0.754729, 1.570796, 1.685284],accel_mss,speed_ms,0,blend_radius_m)
    movel([0.114325, -1.403271, -2.554340, -0.754778, 1.570796, 1.685121],accel_mss,speed_ms,0,blend_radius_m)
    movel([0.114088, -1.403092, -2.554472, -0.754825, 1.570796, 1.684885],accel_mss,speed_ms,0,blend_radius_m)
    movel([0.114422, -1.402771, -2.554709, -0.754909, 1.570796, 1.685218],accel_mss,speed_ms,0,blend_radius_m)
    movel([0.114756, -1.402449, -2.554947, -0.754993, 1.570796, 1.685552],accel_mss,speed_ms,0,blend_radius_m)
    movel([0.114495, -1.402217, -2.555118, -0.755054, 1.570796, 1.685292],accel_mss,speed_ms,0,blend_radius_m)
    movel([0.114323, -1.402013, -2.555268, -0.755108, 1.570796, 1.685119],accel_mss,speed_ms,0,blend_radius_m)
    movel([0.114274, -1.401816, -2.555414, -0.755159, 1.570796, 1.685070],accel_mss,speed_ms,0,blend_radius_m)
    movel([0.114523, -1.401391, -2.555726, -0.755271, 1.570796, 1.685319],accel_mss,speed_ms,0,blend_radius_m)
    movel([0.115063, -1.401146, -2.555907, -0.755336, 1.570796, 1.685859],accel_mss,speed_ms,0,blend_radius_m)
    movel([0.115634, -1.401022, -2.555998, -0.755369, 1.570796, 1.686431],accel_mss,speed_ms,0,blend_radius_m)
    movel([0.116923, -1.400790, -2.556169, -0.755430, 1.570796, 1.687720],accel_mss,speed_ms,0,blend_radius_m)
    speed_ms = 0.003
    movel([0.116923, -1.404026, -2.557622, -0.750741, 1.570796, 1.687720],accel_mss,speed_ms,0,blend_radius_m)
    speed_ms = 0.007
    movel([0.118450, -1.403778, -2.557805, -0.750806, 1.570796, 1.689246],accel_mss,speed_ms,0,blend_radius_m)
    movel([0.119164, -1.403723, -2.557846, -0.750820, 1.570796, 1.689961],accel_mss,speed_ms,0,blend_radius_m)
    movel([0.119522, -1.403808, -2.557783, -0.750798, 1.570796, 1.690318],accel_mss,speed_ms,0,blend_radius_m)
    movel([0.119673, -1.404040, -2.557611, -0.750737, 1.570796, 1.690469],accel_mss,speed_ms,0,blend_radius_m)
    movel([0.119491, -1.404334, -2.557394, -0.750660, 1.570796, 1.690287],accel_mss,speed_ms,0,blend_radius_m)
    movel([0.119212, -1.404740, -2.557094, -0.750555, 1.570796, 1.690008],accel_mss,speed_ms,0,blend_radius_m)
    movel([0.119126, -1.405055, -2.556861, -0.750473, 1.570796, 1.689922],accel_mss,speed_ms,0,blend_radius_m)
    movel([0.119166, -1.405258, -2.556711, -0.750421, 1.570796, 1.689962],accel_mss,speed_ms,0,blend_radius_m)
    movel([0.119206, -1.405459, -2.556562, -0.750369, 1.570796, 1.690002],accel_mss,speed_ms,0,blend_radius_m)
    movel([0.119129, -1.405742, -2.556352, -0.750295, 1.570796, 1.689926],accel_mss,speed_ms,0,blend_radius_m)
    movel([0.118545, -1.406374, -2.555882, -0.750132, 1.570796, 1.689342],accel_mss,speed_ms,0,blend_radius_m)
    movel([0.118026, -1.406708, -2.555634, -0.750046, 1.570796, 1.688823],accel_mss,speed_ms,0,blend_radius_m)
    movel([0.117329, -1.406992, -2.555424, -0.749974, 1.570796, 1.688126],accel_mss,speed_ms,0,blend_radius_m)
    movel([0.116307, -1.407280, -2.555210, -0.749900, 1.570796, 1.687103],accel_mss,speed_ms,0,blend_radius_m)
    movel([0.115098, -1.407542, -2.555014, -0.749833, 1.570796, 1.685894],accel_mss,speed_ms,0,blend_radius_m)
    movel([0.114445, -1.407551, -2.555008, -0.749830, 1.570796, 1.685242],accel_mss,speed_ms,0,blend_radius_m)
    movel([0.114245, -1.407329, -2.555173, -0.749887, 1.570796, 1.685042],accel_mss,speed_ms,0,blend_radius_m)
    movel([0.114389, -1.406920, -2.555477, -0.749992, 1.570796, 1.685185],accel_mss,speed_ms,0,blend_radius_m)
    movel([0.114487, -1.406690, -2.555648, -0.750051, 1.570796, 1.685284],accel_mss,speed_ms,0,blend_radius_m)
    movel([0.114325, -1.406501, -2.555788, -0.750100, 1.570796, 1.685121],accel_mss,speed_ms,0,blend_radius_m)
    movel([0.114088, -1.406322, -2.555921, -0.750146, 1.570796, 1.684885],accel_mss,speed_ms,0,blend_radius_m)
    movel([0.114422, -1.406002, -2.556159, -0.750228, 1.570796, 1.685218],accel_mss,speed_ms,0,blend_radius_m)
    movel([0.114756, -1.405681, -2.556397, -0.750311, 1.570796, 1.685552],accel_mss,speed_ms,0,blend_radius_m)
    movel([0.114495, -1.405449, -2.556569, -0.750371, 1.570796, 1.685292],accel_mss,speed_ms,0,blend_radius_m)
    movel([0.114323, -1.405246, -2.556719, -0.750424, 1.570796, 1.685119],accel_mss,speed_ms,0,blend_radius_m)
    movel([0.114274, -1.405050, -2.556865, -0.750475, 1.570796, 1.685070],accel_mss,speed_ms,0,blend_radius_m)
    movel([0.114523, -1.404626, -2.557178, -0.750585, 1.570796, 1.685319],accel_mss,speed_ms,0,blend_radius_m)
    movel([0.115063, -1.404382, -2.557359, -0.750648, 1.570796, 1.685859],accel_mss,speed_ms,0,blend_radius_m)
    movel([0.115634, -1.404258, -2.557451, -0.750680, 1.570796, 1.686431],accel_mss,speed_ms,0,blend_radius_m)
    movel([0.116923, -1.404026, -2.557622, -0.750741, 1.570796, 1.687720],accel_mss,speed_ms,0,blend_radius_m)
    speed_ms = 0.003
    movel([0.116923, -1.391208, -2.551760, -0.769421, 1.570796, 1.687720],accel_mss,speed_ms,0,blend_radius_m)
    speed_ms = 1.000
    movel([0.116923, -1.366587, -2.539643, -0.806159, 1.570796, 1.687720],accel_mss,speed_ms,0,blend_radius_m)
    movel([0.116275, -1.370444, -2.536938, -0.805007, 1.570796, 1.687072],accel_mss,speed_ms,0,blend_radius_m)
    movel([0.116275, -1.394993, -2.549006, -0.768389, 1.570796, 1.687072],accel_mss,speed_ms,0,blend_radius_m)
    speed_ms = 0.003
    movel([0.116275, -1.404545, -2.553397, -0.754447, 1.570796, 1.687072],accel_mss,speed_ms,0,blend_radius_m)
    speed_ms = 0.007
    movel([0.116705, -1.404434, -2.553479, -0.754476, 1.570796, 1.687501],accel_mss,speed_ms,0,blend_radius_m)
    movel([0.117062, -1.404455, -2.553464, -0.754470, 1.570796, 1.687859],accel_mss,speed_ms,0,blend_radius_m)
    movel([0.117167, -1.404617, -2.553344, -0.754428, 1.570796, 1.687963],accel_mss,speed_ms,0,blend_radius_m)
    movel([0.116942, -1.404907, -2.553129, -0.754353, 1.570796, 1.687739],accel_mss,speed_ms,0,blend_radius_m)
    movel([0.116708, -1.405086, -2.552996, -0.754307, 1.570796, 1.687504],accel_mss,speed_ms,0,blend_radius_m)
    movel([0.116444, -1.405186, -2.552922, -0.754281, 1.570796, 1.687240],accel_mss,speed_ms,0,blend_radius_m)
    movel([0.116190, -1.405195, -2.552915, -0.754279, 1.570796, 1.686986],accel_mss,speed_ms,0,blend_radius_m)
    movel([0.115991, -1.405108, -2.552980, -0.754301, 1.570796, 1.686788],accel_mss,speed_ms,0,blend_radius_m)
    movel([0.115873, -1.404946, -2.553100, -0.754343, 1.570796, 1.686669],accel_mss,speed_ms,0,blend_radius_m)
    movel([0.116275, -1.404545, -2.553397, -0.754447, 1.570796, 1.687072],accel_mss,speed_ms,0,blend_radius_m)
    speed_ms = 0.003
    movel([0.116275, -1.407771, -2.554844, -0.749774, 1.570796, 1.687072],accel_mss,speed_ms,0,blend_radius_m)
    speed_ms = 0.007
    movel([0.116705, -1.407660, -2.554926, -0.749802, 1.570796, 1.687501],accel_mss,speed_ms,0,blend_radius_m)
    movel([0.117062, -1.407681, -2.554911, -0.749797, 1.570796, 1.687859],accel_mss,speed_ms,0,blend_radius_m)
    movel([0.117167, -1.407843, -2.554790, -0.749756, 1.570796, 1.687963],accel_mss,speed_ms,0,blend_radius_m)
    movel([0.116942, -1.408132, -2.554575, -0.749682, 1.570796, 1.687739],accel_mss,speed_ms,0,blend_radius_m)
    movel([0.116708, -1.408311, -2.554442, -0.749637, 1.570796, 1.687504],accel_mss,speed_ms,0,blend_radius_m)
    movel([0.116444, -1.408410, -2.554368, -0.749611, 1.570796, 1.687240],accel_mss,speed_ms,0,blend_radius_m)
    movel([0.116190, -1.408420, -2.554361, -0.749609, 1.570796, 1.686986],accel_mss,speed_ms,0,blend_radius_m)
    movel([0.115991, -1.408333, -2.554425, -0.749631, 1.570796, 1.686788],accel_mss,speed_ms,0,blend_radius_m)
    movel([0.115873, -1.408171, -2.554546, -0.749672, 1.570796, 1.686669],accel_mss,speed_ms,0,blend_radius_m)
    movel([0.116275, -1.407771, -2.554844, -0.749774, 1.570796, 1.687072],accel_mss,speed_ms,0,blend_radius_m)
    speed_ms = 0.003
    movel([0.116275, -1.394993, -2.549006, -0.768389, 1.570796, 1.687072],accel_mss,speed_ms,0,blend_radius_m)
    speed_ms = 1.000
    movel([0.116275, -1.370444, -2.536938, -0.805007, 1.570796, 1.687072],accel_mss,speed_ms,0,blend_radius_m)
    movel([0.071617, -1.356963, -2.546304, -0.809122, 1.570796, 1.642413],accel_mss,speed_ms,0,blend_radius_m)
    movel([0.071617, -1.381761, -2.558542, -0.772086, 1.570796, 1.642413],accel_mss,speed_ms,0,blend_radius_m)
    speed_ms = 0.003
    movel([0.071617, -1.391418, -2.562997, -0.757974, 1.570796, 1.642413],accel_mss,speed_ms,0,blend_radius_m)
    speed_ms = 0.007
    movel([0.069577, -1.391884, -2.562661, -0.757845, 1.570796, 1.640373],accel_mss,speed_ms,0,blend_radius_m)
    movel([0.068922, -1.391989, -2.562584, -0.757815, 1.570796, 1.639718],accel_mss,speed_ms,0,blend_radius_m)
    movel([0.068598, -1.391994, -2.562581, -0.757814, 1.570796, 1.639395],accel_mss,speed_ms,0,blend_radius_m)
    movel([0.068461, -1.391838, -2.562694, -0.757857, 1.570796, 1.639258],accel_mss,speed_ms,0,blend_radius_m)
    movel([0.068638, -1.391563, -2.562892, -0.757934, 1.570796, 1.639434],accel_mss,speed_ms,0,blend_radius_m)
    movel([0.069122, -1.391247, -2.563120, -0.758022, 1.570796, 1.639918],accel_mss,speed_ms,0,blend_radius_m)
    movel([0.070213, -1.390930, -2.563349, -0.758110, 1.570796, 1.641009],accel_mss,speed_ms,0,blend_radius_m)
    movel([0.071290, -1.390711, -2.563507, -0.758171, 1.570796, 1.642087],accel_mss,speed_ms,0,blend_radius_m)
    movel([0.071672, -1.390815, -2.563432, -0.758142, 1.570796, 1.642469],accel_mss,speed_ms,0,blend_radius_m)
    movel([0.071727, -1.391083, -2.563239, -0.758068, 1.570796, 1.642523],accel_mss,speed_ms,0,blend_radius_m)
    movel([0.071675, -1.391329, -2.563061, -0.757999, 1.570796, 1.642471],accel_mss,speed_ms,0,blend_radius_m)
    speed_ms = 0.003
    movel([0.071617, -1.394681, -2.564465, -0.753243, 1.570796, 1.642413],accel_mss,speed_ms,0,blend_radius_m)
    speed_ms = 0.007
    movel([0.069577, -1.395145, -2.564128, -0.753116, 1.570796, 1.640373],accel_mss,speed_ms,0,blend_radius_m)
    movel([0.068922, -1.395251, -2.564051, -0.753087, 1.570796, 1.639718],accel_mss,speed_ms,0,blend_radius_m)
    movel([0.068598, -1.395255, -2.564048, -0.753086, 1.570796, 1.639395],accel_mss,speed_ms,0,blend_radius_m)
    movel([0.068461, -1.395099, -2.564161, -0.753129, 1.570796, 1.639258],accel_mss,speed_ms,0,blend_radius_m)
    movel([0.068638, -1.394825, -2.564360, -0.753204, 1.570796, 1.639434],accel_mss,speed_ms,0,blend_radius_m)
    movel([0.069122, -1.394510, -2.564589, -0.753290, 1.570796, 1.639918],accel_mss,speed_ms,0,blend_radius_m)
    movel([0.070213, -1.394194, -2.564818, -0.753377, 1.570796, 1.641009],accel_mss,speed_ms,0,blend_radius_m)
    movel([0.071290, -1.393975, -2.564976, -0.753438, 1.570796, 1.642087],accel_mss,speed_ms,0,blend_radius_m)
    movel([0.071672, -1.394079, -2.564901, -0.753409, 1.570796, 1.642469],accel_mss,speed_ms,0,blend_radius_m)
    movel([0.071727, -1.394346, -2.564707, -0.753335, 1.570796, 1.642523],accel_mss,speed_ms,0,blend_radius_m)
    movel([0.071675, -1.394592, -2.564529, -0.753268, 1.570796, 1.642471],accel_mss,speed_ms,0,blend_radius_m)
    speed_ms = 0.003
    movel([0.071617, -1.381761, -2.558542, -0.772086, 1.570796, 1.642413],accel_mss,speed_ms,0,blend_radius_m)
    speed_ms = 1.000
    movel([0.071617, -1.356963, -2.546304, -0.809122, 1.570796, 1.642413],accel_mss,speed_ms,0,blend_radius_m)
    movel([0.071390, -1.355193, -2.547515, -0.809680, 1.570796, 1.642186],accel_mss,speed_ms,0,blend_radius_m)
    movel([0.071390, -1.380023, -2.559776, -0.772590, 1.570796, 1.642186],accel_mss,speed_ms,0,blend_radius_m)
    speed_ms = 0.003
    movel([0.071390, -1.389694, -2.564239, -0.758456, 1.570796, 1.642186],accel_mss,speed_ms,0,blend_radius_m)
    speed_ms = 0.007
    movel([0.071125, -1.389804, -2.564160, -0.758425, 1.570796, 1.641921],accel_mss,speed_ms,0,blend_radius_m)
    movel([0.070507, -1.389824, -2.564145, -0.758420, 1.570796, 1.641303],accel_mss,speed_ms,0,blend_radius_m)
    movel([0.069879, -1.389788, -2.564171, -0.758430, 1.570796, 1.640675],accel_mss,speed_ms,0,blend_radius_m)
    movel([0.069421, -1.389680, -2.564249, -0.758460, 1.570796, 1.640217],accel_mss,speed_ms,0,blend_radius_m)
    movel([0.068816, -1.389330, -2.564501, -0.758558, 1.570796, 1.639612],accel_mss,speed_ms,0,blend_radius_m)
    movel([0.068448, -1.388813, -2.564872, -0.758704, 1.570796, 1.639245],accel_mss,speed_ms,0,blend_radius_m)
    movel([0.068281, -1.388058, -2.565413, -0.758917, 1.570796, 1.639078],accel_mss,speed_ms,0,blend_radius_m)
    movel([0.068297, -1.386960, -2.566200, -0.759229, 1.570796, 1.639093],accel_mss,speed_ms,0,blend_radius_m)
    movel([0.068504, -1.385834, -2.567004, -0.759551, 1.570796, 1.639300],accel_mss,speed_ms,0,blend_radius_m)
    movel([0.068940, -1.384856, -2.567702, -0.759832, 1.570796, 1.639736],accel_mss,speed_ms,0,blend_radius_m)
    movel([0.069611, -1.384023, -2.568295, -0.760072, 1.570796, 1.640407],accel_mss,speed_ms,0,blend_radius_m)
    movel([0.070503, -1.383332, -2.568785, -0.760272, 1.570796, 1.641299],accel_mss,speed_ms,0,blend_radius_m)
    movel([0.071108, -1.383026, -2.569002, -0.760360, 1.570796, 1.641904],accel_mss,speed_ms,0,blend_radius_m)
    movel([0.071382, -1.383068, -2.568972, -0.760348, 1.570796, 1.642178],accel_mss,speed_ms,0,blend_radius_m)
    movel([0.071487, -1.383440, -2.568708, -0.760240, 1.570796, 1.642283],accel_mss,speed_ms,0,blend_radius_m)
    movel([0.071463, -1.384769, -2.567763, -0.759856, 1.570796, 1.642260],accel_mss,speed_ms,0,blend_radius_m)
    movel([0.071447, -1.385513, -2.567233, -0.759643, 1.570796, 1.642243],accel_mss,speed_ms,0,blend_radius_m)
    movel([0.071447, -1.386326, -2.566653, -0.759410, 1.570796, 1.642243],accel_mss,speed_ms,0,blend_radius_m)
    movel([0.071456, -1.387087, -2.566109, -0.759193, 1.570796, 1.642252],accel_mss,speed_ms,0,blend_radius_m)
    movel([0.071478, -1.387656, -2.565702, -0.759031, 1.570796, 1.642275],accel_mss,speed_ms,0,blend_radius_m)
    movel([0.071526, -1.388621, -2.565010, -0.758758, 1.570796, 1.642322],accel_mss,speed_ms,0,blend_radius_m)
    movel([0.071525, -1.389181, -2.564608, -0.758600, 1.570796, 1.642321],accel_mss,speed_ms,0,blend_radius_m)
    movel([0.071490, -1.389540, -2.564349, -0.758499, 1.570796, 1.642286],accel_mss,speed_ms,0,blend_radius_m)
    speed_ms = 0.003
    movel([0.071390, -1.392961, -2.565710, -0.753718, 1.570796, 1.642186],accel_mss,speed_ms,0,blend_radius_m)
    speed_ms = 0.007
    movel([0.071125, -1.393071, -2.565630, -0.753687, 1.570796, 1.641921],accel_mss,speed_ms,0,blend_radius_m)
    movel([0.070507, -1.393091, -2.565616, -0.753682, 1.570796, 1.641303],accel_mss,speed_ms,0,blend_radius_m)
    movel([0.069879, -1.393055, -2.565642, -0.753692, 1.570796, 1.640675],accel_mss,speed_ms,0,blend_radius_m)
    movel([0.069421, -1.392947, -2.565720, -0.753722, 1.570796, 1.640217],accel_mss,speed_ms,0,blend_radius_m)
    movel([0.068816, -1.392599, -2.565972, -0.753819, 1.570796, 1.639612],accel_mss,speed_ms,0,blend_radius_m)
    movel([0.068448, -1.392083, -2.566344, -0.753962, 1.570796, 1.639245],accel_mss,speed_ms,0,blend_radius_m)
    movel([0.068281, -1.391330, -2.566887, -0.754172, 1.570796, 1.639078],accel_mss,speed_ms,0,blend_radius_m)
    movel([0.068297, -1.390235, -2.567675, -0.754479, 1.570796, 1.639093],accel_mss,speed_ms,0,blend_radius_m)
    movel([0.068504, -1.389112, -2.568481, -0.754795, 1.570796, 1.639300],accel_mss,speed_ms,0,blend_radius_m)
    movel([0.068940, -1.388136, -2.569181, -0.755072, 1.570796, 1.639736],accel_mss,speed_ms,0,blend_radius_m)
    movel([0.069611, -1.387306, -2.569775, -0.755309, 1.570796, 1.640407],accel_mss,speed_ms,0,blend_radius_m)
    movel([0.070503, -1.386617, -2.570266, -0.755506, 1.570796, 1.641299],accel_mss,speed_ms,0,blend_radius_m)
    movel([0.071108, -1.386312, -2.570484, -0.755593, 1.570796, 1.641904],accel_mss,speed_ms,0,blend_radius_m)
    movel([0.071382, -1.386354, -2.570454, -0.755581, 1.570796, 1.642178],accel_mss,speed_ms,0,blend_radius_m)
    movel([0.071487, -1.386725, -2.570189, -0.755475, 1.570796, 1.642283],accel_mss,speed_ms,0,blend_radius_m)
    movel([0.071463, -1.388050, -2.569242, -0.755097, 1.570796, 1.642260],accel_mss,speed_ms,0,blend_radius_m)
    movel([0.071447, -1.388792, -2.568711, -0.754886, 1.570796, 1.642243],accel_mss,speed_ms,0,blend_radius_m)
    movel([0.071447, -1.389603, -2.568129, -0.754657, 1.570796, 1.642243],accel_mss,speed_ms,0,blend_radius_m)
    movel([0.071456, -1.390362, -2.567584, -0.754443, 1.570796, 1.642252],accel_mss,speed_ms,0,blend_radius_m)
    movel([0.071478, -1.390929, -2.567176, -0.754284, 1.570796, 1.642275],accel_mss,speed_ms,0,blend_radius_m)
    movel([0.071526, -1.391892, -2.566482, -0.754015, 1.570796, 1.642322],accel_mss,speed_ms,0,blend_radius_m)
    movel([0.071525, -1.392450, -2.566079, -0.753860, 1.570796, 1.642321],accel_mss,speed_ms,0,blend_radius_m)
    movel([0.071490, -1.392808, -2.565821, -0.753760, 1.570796, 1.642286],accel_mss,speed_ms,0,blend_radius_m)
    speed_ms = 0.003
    movel([0.071390, -1.380023, -2.559776, -0.772590, 1.570796, 1.642186],accel_mss,speed_ms,0,blend_radius_m)
    speed_ms = 1.000
    movel([0.071390, -1.355193, -2.547515, -0.809680, 1.570796, 1.642186],accel_mss,speed_ms,0,blend_radius_m)
    movel([0.064153, -1.352173, -2.549573, -0.810644, 1.570796, 1.634949],accel_mss,speed_ms,0,blend_radius_m)
    movel([0.064153, -1.377057, -2.561872, -0.773460, 1.570796, 1.634949],accel_mss,speed_ms,0,blend_radius_m)
    speed_ms = 0.003
    movel([0.064153, -1.386751, -2.566349, -0.759289, 1.570796, 1.634949],accel_mss,speed_ms,0,blend_radius_m)
    speed_ms = 0.007
    movel([0.063340, -1.387772, -2.565619, -0.758999, 1.570796, 1.634136],accel_mss,speed_ms,0,blend_radius_m)
    movel([0.062686, -1.388569, -2.565047, -0.758773, 1.570796, 1.633482],accel_mss,speed_ms,0,blend_radius_m)
    movel([0.062675, -1.388124, -2.565366, -0.758899, 1.570796, 1.633471],accel_mss,speed_ms,0,blend_radius_m)
    movel([0.062900, -1.387745, -2.565638, -0.759006, 1.570796, 1.633696],accel_mss,speed_ms,0,blend_radius_m)
    movel([0.063169, -1.387429, -2.565864, -0.759096, 1.570796, 1.633965],accel_mss,speed_ms,0,blend_radius_m)
    movel([0.063443, -1.387047, -2.566137, -0.759204, 1.570796, 1.634239],accel_mss,speed_ms,0,blend_radius_m)
    movel([0.063524, -1.386809, -2.566308, -0.759272, 1.570796, 1.634320],accel_mss,speed_ms,0,blend_radius_m)
    movel([0.063593, -1.386471, -2.566549, -0.759368, 1.570796, 1.634389],accel_mss,speed_ms,0,blend_radius_m)
    movel([0.063654, -1.386177, -2.566759, -0.759452, 1.570796, 1.634450],accel_mss,speed_ms,0,blend_radius_m)
    movel([0.063753, -1.385826, -2.567010, -0.759553, 1.570796, 1.634549],accel_mss,speed_ms,0,blend_radius_m)
    movel([0.063869, -1.385475, -2.567261, -0.759654, 1.570796, 1.634666],accel_mss,speed_ms,0,blend_radius_m)
    movel([0.063989, -1.385181, -2.567470, -0.759738, 1.570796, 1.634785],accel_mss,speed_ms,0,blend_radius_m)
    movel([0.064155, -1.384750, -2.567777, -0.759862, 1.570796, 1.634951],accel_mss,speed_ms,0,blend_radius_m)
    movel([0.064180, -1.384485, -2.567966, -0.759938, 1.570796, 1.634976],accel_mss,speed_ms,0,blend_radius_m)
    movel([0.063844, -1.384381, -2.568040, -0.759968, 1.570796, 1.634641],accel_mss,speed_ms,0,blend_radius_m)
    movel([0.063665, -1.384201, -2.568168, -0.760020, 1.570796, 1.634461],accel_mss,speed_ms,0,blend_radius_m)
    movel([0.063664, -1.383761, -2.568481, -0.760147, 1.570796, 1.634460],accel_mss,speed_ms,0,blend_radius_m)
    movel([0.063663, -1.383539, -2.568639, -0.760212, 1.570796, 1.634460],accel_mss,speed_ms,0,blend_radius_m)
    movel([0.063659, -1.383178, -2.568894, -0.760316, 1.570796, 1.634455],accel_mss,speed_ms,0,blend_radius_m)
    movel([0.063652, -1.382770, -2.569184, -0.760435, 1.570796, 1.634449],accel_mss,speed_ms,0,blend_radius_m)
    movel([0.063644, -1.382363, -2.569473, -0.760553, 1.570796, 1.634440],accel_mss,speed_ms,0,blend_radius_m)
    movel([0.063647, -1.381532, -2.570061, -0.760796, 1.570796, 1.634444],accel_mss,speed_ms,0,blend_radius_m)
    movel([0.063692, -1.380836, -2.570553, -0.761000, 1.570796, 1.634488],accel_mss,speed_ms,0,blend_radius_m)
    movel([0.063775, -1.380285, -2.570942, -0.761162, 1.570796, 1.634571],accel_mss,speed_ms,0,blend_radius_m)
    movel([0.063897, -1.379969, -2.571165, -0.761255, 1.570796, 1.634693],accel_mss,speed_ms,0,blend_radius_m)
    movel([0.064290, -1.379690, -2.571361, -0.761337, 1.570796, 1.635086],accel_mss,speed_ms,0,blend_radius_m)
    movel([0.064739, -1.379526, -2.571477, -0.761386, 1.570796, 1.635535],accel_mss,speed_ms,0,blend_radius_m)
    movel([0.065708, -1.379220, -2.571693, -0.761476, 1.570796, 1.636505],accel_mss,speed_ms,0,blend_radius_m)
    movel([0.066539, -1.378970, -2.571869, -0.761550, 1.570796, 1.637335],accel_mss,speed_ms,0,blend_radius_m)
    movel([0.067034, -1.378840, -2.571960, -0.761589, 1.570796, 1.637831],accel_mss,speed_ms,0,blend_radius_m)
    movel([0.067345, -1.378784, -2.571999, -0.761605, 1.570796, 1.638141],accel_mss,speed_ms,0,blend_radius_m)
    movel([0.067187, -1.379390, -2.571573, -0.761426, 1.570796, 1.637983],accel_mss,speed_ms,0,blend_radius_m)
    movel([0.066879, -1.379944, -2.571182, -0.761262, 1.570796, 1.637675],accel_mss,speed_ms,0,blend_radius_m)
    movel([0.066506, -1.380579, -2.570734, -0.761075, 1.570796, 1.637303],accel_mss,speed_ms,0,blend_radius_m)
    movel([0.066134, -1.381213, -2.570286, -0.760889, 1.570796, 1.636931],accel_mss,speed_ms,0,blend_radius_m)
    movel([0.065832, -1.381769, -2.569893, -0.760727, 1.570796, 1.636628],accel_mss,speed_ms,0,blend_radius_m)
    movel([0.065596, -1.382232, -2.569566, -0.760592, 1.570796, 1.636392],accel_mss,speed_ms,0,blend_radius_m)
    movel([0.065843, -1.382380, -2.569460, -0.760548, 1.570796, 1.636640],accel_mss,speed_ms,0,blend_radius_m)
    movel([0.066139, -1.382317, -2.569505, -0.760567, 1.570796, 1.636935],accel_mss,speed_ms,0,blend_radius_m)
    movel([0.066626, -1.382174, -2.569607, -0.760609, 1.570796, 1.637423],accel_mss,speed_ms,0,blend_radius_m)
    movel([0.067199, -1.382006, -2.569725, -0.760657, 1.570796, 1.637995],accel_mss,speed_ms,0,blend_radius_m)
    movel([0.067529, -1.381937, -2.569775, -0.760678, 1.570796, 1.638325],accel_mss,speed_ms,0,blend_radius_m)
    movel([0.067763, -1.382007, -2.569725, -0.760657, 1.570796, 1.638559],accel_mss,speed_ms,0,blend_radius_m)
    movel([0.067012, -1.383013, -2.569012, -0.760364, 1.570796, 1.637808],accel_mss,speed_ms,0,blend_radius_m)
    movel([0.066191, -1.384094, -2.568244, -0.760051, 1.570796, 1.636988],accel_mss,speed_ms,0,blend_radius_m)
    movel([0.065221, -1.385365, -2.567339, -0.759685, 1.570796, 1.636018],accel_mss,speed_ms,0,blend_radius_m)
    movel([0.064153, -1.386751, -2.566349, -0.759289, 1.570796, 1.634949],accel_mss,speed_ms,0,blend_radius_m)
    speed_ms = 0.003
    movel([0.064153, -1.390026, -2.567825, -0.754538, 1.570796, 1.634949],accel_mss,speed_ms,0,blend_radius_m)
    speed_ms = 0.007
    movel([0.063340, -1.391044, -2.567093, -0.754252, 1.570796, 1.634136],accel_mss,speed_ms,0,blend_radius_m)
    movel([0.062686, -1.391840, -2.566520, -0.754030, 1.570796, 1.633482],accel_mss,speed_ms,0,blend_radius_m)
    movel([0.062675, -1.391396, -2.566839, -0.754153, 1.570796, 1.633471],accel_mss,speed_ms,0,blend_radius_m)
    movel([0.062900, -1.391018, -2.567112, -0.754259, 1.570796, 1.633696],accel_mss,speed_ms,0,blend_radius_m)
    movel([0.063169, -1.390703, -2.567339, -0.754348, 1.570796, 1.633965],accel_mss,speed_ms,0,blend_radius_m)
    movel([0.063443, -1.390322, -2.567612, -0.754454, 1.570796, 1.634239],accel_mss,speed_ms,0,blend_radius_m)
    movel([0.063524, -1.390085, -2.567783, -0.754521, 1.570796, 1.634320],accel_mss,speed_ms,0,blend_radius_m)
    movel([0.063593, -1.389748, -2.568025, -0.754616, 1.570796, 1.634389],accel_mss,speed_ms,0,blend_radius_m)
    movel([0.063654, -1.389454, -2.568236, -0.754699, 1.570796, 1.634450],accel_mss,speed_ms,0,blend_radius_m)
    movel([0.063753, -1.389104, -2.568487, -0.754798, 1.570796, 1.634549],accel_mss,speed_ms,0,blend_radius_m)
    movel([0.063869, -1.388754, -2.568738, -0.754897, 1.570796, 1.634666],accel_mss,speed_ms,0,blend_radius_m)
    movel([0.063989, -1.388461, -2.568948, -0.754980, 1.570796, 1.634785],accel_mss,speed_ms,0,blend_radius_m)
    movel([0.064155, -1.388031, -2.569256, -0.755102, 1.570796, 1.634951],accel_mss,speed_ms,0,blend_radius_m)
    movel([0.064180, -1.387767, -2.569445, -0.755177, 1.570796, 1.634976],accel_mss,speed_ms,0,blend_radius_m)
    movel([0.063844, -1.387663, -2.569519, -0.755207, 1.570796, 1.634641],accel_mss,speed_ms,0,blend_radius_m)
    movel([0.063665, -1.387484, -2.569647, -0.755258, 1.570796, 1.634461],accel_mss,speed_ms,0,blend_radius_m)
    movel([0.063664, -1.387045, -2.569961, -0.755383, 1.570796, 1.634460],accel_mss,speed_ms,0,blend_radius_m)
    movel([0.063663, -1.386823, -2.570119, -0.755447, 1.570796, 1.634460],accel_mss,speed_ms,0,blend_radius_m)
    movel([0.063659, -1.386464, -2.570376, -0.755550, 1.570796, 1.634455],accel_mss,speed_ms,0,blend_radius_m)
    movel([0.063652, -1.386057, -2.570666, -0.755666, 1.570796, 1.634449],accel_mss,speed_ms,0,blend_radius_m)
    movel([0.063644, -1.385650, -2.570956, -0.755783, 1.570796, 1.634440],accel_mss,speed_ms,0,blend_radius_m)
    movel([0.063647, -1.384822, -2.571545, -0.756022, 1.570796, 1.634444],accel_mss,speed_ms,0,blend_radius_m)
    movel([0.063692, -1.384128, -2.572038, -0.756223, 1.570796, 1.634488],accel_mss,speed_ms,0,blend_radius_m)
    movel([0.063775, -1.383578, -2.572429, -0.756383, 1.570796, 1.634571],accel_mss,speed_ms,0,blend_radius_m)
    movel([0.063897, -1.383263, -2.572652, -0.756474, 1.570796, 1.634693],accel_mss,speed_ms,0,blend_radius_m)
    movel([0.064290, -1.382985, -2.572849, -0.756555, 1.570796, 1.635086],accel_mss,speed_ms,0,blend_radius_m)
    movel([0.064739, -1.382821, -2.572964, -0.756603, 1.570796, 1.635535],accel_mss,speed_ms,0,blend_radius_m)
    movel([0.065708, -1.382516, -2.573181, -0.756692, 1.570796, 1.636505],accel_mss,speed_ms,0,blend_radius_m)
    movel([0.066539, -1.382267, -2.573357, -0.756765, 1.570796, 1.637335],accel_mss,speed_ms,0,blend_radius_m)
    movel([0.067034, -1.382137, -2.573449, -0.756803, 1.570796, 1.637831],accel_mss,speed_ms,0,blend_radius_m)
    movel([0.067345, -1.382082, -2.573488, -0.756819, 1.570796, 1.638141],accel_mss,speed_ms,0,blend_radius_m)
    movel([0.067187, -1.382685, -2.573061, -0.756643, 1.570796, 1.637983],accel_mss,speed_ms,0,blend_radius_m)
    movel([0.066879, -1.383239, -2.572669, -0.756481, 1.570796, 1.637675],accel_mss,speed_ms,0,blend_radius_m)
    movel([0.066506, -1.383872, -2.572220, -0.756297, 1.570796, 1.637303],accel_mss,speed_ms,0,blend_radius_m)
    movel([0.066134, -1.384504, -2.571771, -0.756114, 1.570796, 1.636931],accel_mss,speed_ms,0,blend_radius_m)
    movel([0.065832, -1.385059, -2.571377, -0.755954, 1.570796, 1.636628],accel_mss,speed_ms,0,blend_radius_m)
    movel([0.065596, -1.385520, -2.571049, -0.755821, 1.570796, 1.636392],accel_mss,speed_ms,0,blend_radius_m)
    movel([0.065843, -1.385668, -2.570943, -0.755778, 1.570796, 1.636640],accel_mss,speed_ms,0,blend_radius_m)
    movel([0.066139, -1.385605, -2.570988, -0.755796, 1.570796, 1.636935],accel_mss,speed_ms,0,blend_radius_m)
    movel([0.066626, -1.385462, -2.571090, -0.755837, 1.570796, 1.637423],accel_mss,speed_ms,0,blend_radius_m)
    movel([0.067199, -1.385295, -2.571209, -0.755885, 1.570796, 1.637995],accel_mss,speed_ms,0,blend_radius_m)
    movel([0.067529, -1.385225, -2.571258, -0.755906, 1.570796, 1.638325],accel_mss,speed_ms,0,blend_radius_m)
    movel([0.067763, -1.385295, -2.571208, -0.755885, 1.570796, 1.638559],accel_mss,speed_ms,0,blend_radius_m)
    movel([0.067012, -1.386299, -2.570493, -0.755597, 1.570796, 1.637808],accel_mss,speed_ms,0,blend_radius_m)
    movel([0.066191, -1.387377, -2.569724, -0.755288, 1.570796, 1.636988],accel_mss,speed_ms,0,blend_radius_m)
    movel([0.065221, -1.388644, -2.568817, -0.754928, 1.570796, 1.636018],accel_mss,speed_ms,0,blend_radius_m)
    movel([0.064153, -1.390026, -2.567825, -0.754538, 1.570796, 1.634949],accel_mss,speed_ms,0,blend_radius_m)
    speed_ms = 0.003
    movel([0.064153, -1.377057, -2.561872, -0.773460, 1.570796, 1.634949],accel_mss,speed_ms,0,blend_radius_m)
    speed_ms = 1.000
    movel([0.064153, -1.352173, -2.549573, -0.810644, 1.570796, 1.634949],accel_mss,speed_ms,0,blend_radius_m)
    movel([0.065962, -1.340154, -2.557638, -0.814597, 1.570796, 1.636759],accel_mss,speed_ms,0,blend_radius_m)
    movel([0.065962, -1.365252, -2.570091, -0.777046, 1.570796, 1.636759],accel_mss,speed_ms,0,blend_radius_m)
    speed_ms = 0.003
    movel([0.065962, -1.375037, -2.574625, -0.762726, 1.570796, 1.636759],accel_mss,speed_ms,0,blend_radius_m)
    speed_ms = 0.007
    movel([0.065737, -1.374802, -2.574789, -0.762797, 1.570796, 1.636533],accel_mss,speed_ms,0,blend_radius_m)
    movel([0.065748, -1.374108, -2.575274, -0.763008, 1.570796, 1.636545],accel_mss,speed_ms,0,blend_radius_m)
    movel([0.065782, -1.373380, -2.575780, -0.763229, 1.570796, 1.636578],accel_mss,speed_ms,0,blend_radius_m)
    movel([0.066186, -1.373075, -2.575992, -0.763321, 1.570796, 1.636982],accel_mss,speed_ms,0,blend_radius_m)
    movel([0.067252, -1.372821, -2.576169, -0.763399, 1.570796, 1.638048],accel_mss,speed_ms,0,blend_radius_m)
    movel([0.068316, -1.372596, -2.576325, -0.763467, 1.570796, 1.639113],accel_mss,speed_ms,0,blend_radius_m)
    movel([0.068585, -1.372629, -2.576302, -0.763457, 1.570796, 1.639381],accel_mss,speed_ms,0,blend_radius_m)
    movel([0.068684, -1.372934, -2.576090, -0.763364, 1.570796, 1.639480],accel_mss,speed_ms,0,blend_radius_m)
    movel([0.068626, -1.373256, -2.575866, -0.763266, 1.570796, 1.639422],accel_mss,speed_ms,0,blend_radius_m)
    movel([0.068470, -1.373815, -2.575478, -0.763096, 1.570796, 1.639267],accel_mss,speed_ms,0,blend_radius_m)
    movel([0.068277, -1.374079, -2.575293, -0.763016, 1.570796, 1.639073],accel_mss,speed_ms,0,blend_radius_m)
    movel([0.067750, -1.374381, -2.575083, -0.762925, 1.570796, 1.638546],accel_mss,speed_ms,0,blend_radius_m)
    movel([0.067148, -1.374646, -2.574898, -0.762845, 1.570796, 1.637944],accel_mss,speed_ms,0,blend_radius_m)
    movel([0.066517, -1.374873, -2.574740, -0.762776, 1.570796, 1.637313],accel_mss,speed_ms,0,blend_radius_m)
    movel([0.065962, -1.375037, -2.574625, -0.762726, 1.570796, 1.636759],accel_mss,speed_ms,0,blend_radius_m)
    speed_ms = 0.003
    movel([0.065962, -1.378345, -2.576120, -0.757924, 1.570796, 1.636759],accel_mss,speed_ms,0,blend_radius_m)
    speed_ms = 0.007
    movel([0.065737, -1.378110, -2.576285, -0.757994, 1.570796, 1.636533],accel_mss,speed_ms,0,blend_radius_m)
    movel([0.065748, -1.377418, -2.576770, -0.758201, 1.570796, 1.636545],accel_mss,speed_ms,0,blend_radius_m)
    movel([0.065782, -1.376692, -2.577278, -0.758419, 1.570796, 1.636578],accel_mss,speed_ms,0,blend_radius_m)
    movel([0.066186, -1.376388, -2.577490, -0.758511, 1.570796, 1.636982],accel_mss,speed_ms,0,blend_radius_m)
    movel([0.067252, -1.376135, -2.577667, -0.758587, 1.570796, 1.638048],accel_mss,speed_ms,0,blend_radius_m)
    movel([0.068316, -1.375910, -2.577824, -0.758655, 1.570796, 1.639113],accel_mss,speed_ms,0,blend_radius_m)
    movel([0.068585, -1.375943, -2.577801, -0.758645, 1.570796, 1.639381],accel_mss,speed_ms,0,blend_radius_m)
    movel([0.068684, -1.376248, -2.577588, -0.758553, 1.570796, 1.639480],accel_mss,speed_ms,0,blend_radius_m)
    movel([0.068626, -1.376569, -2.577364, -0.758456, 1.570796, 1.639422],accel_mss,speed_ms,0,blend_radius_m)
    movel([0.068470, -1.377126, -2.576974, -0.758289, 1.570796, 1.639267],accel_mss,speed_ms,0,blend_radius_m)
    movel([0.068277, -1.377389, -2.576790, -0.758210, 1.570796, 1.639073],accel_mss,speed_ms,0,blend_radius_m)
    movel([0.067750, -1.377691, -2.576579, -0.758120, 1.570796, 1.638546],accel_mss,speed_ms,0,blend_radius_m)
    movel([0.067148, -1.377954, -2.576394, -0.758041, 1.570796, 1.637944],accel_mss,speed_ms,0,blend_radius_m)
    movel([0.066517, -1.378181, -2.576235, -0.757973, 1.570796, 1.637313],accel_mss,speed_ms,0,blend_radius_m)
    movel([0.065962, -1.378345, -2.576120, -0.757924, 1.570796, 1.636759],accel_mss,speed_ms,0,blend_radius_m)
    speed_ms = 0.003
    movel([0.065962, -1.365252, -2.570091, -0.777046, 1.570796, 1.636759],accel_mss,speed_ms,0,blend_radius_m)
    speed_ms = 1.000
    movel([0.065962, -1.340154, -2.557638, -0.814597, 1.570796, 1.636759],accel_mss,speed_ms,0,blend_radius_m)
    movel([0.067314, -1.337303, -2.559523, -0.815563, 1.570796, 1.638110],accel_mss,speed_ms,0,blend_radius_m)
    movel([0.067314, -1.362450, -2.572012, -0.777926, 1.570796, 1.638110],accel_mss,speed_ms,0,blend_radius_m)
    speed_ms = 0.003
    movel([0.067314, -1.372257, -2.576561, -0.763571, 1.570796, 1.638110],accel_mss,speed_ms,0,blend_radius_m)
    speed_ms = 0.007
    movel([0.067188, -1.372005, -2.576736, -0.763648, 1.570796, 1.637984],accel_mss,speed_ms,0,blend_radius_m)
    movel([0.067191, -1.371585, -2.577027, -0.763777, 1.570796, 1.637988],accel_mss,speed_ms,0,blend_radius_m)
    movel([0.067248, -1.370744, -2.577609, -0.764035, 1.570796, 1.638044],accel_mss,speed_ms,0,blend_radius_m)
    movel([0.067309, -1.370030, -2.578103, -0.764256, 1.570796, 1.638105],accel_mss,speed_ms,0,blend_radius_m)
    movel([0.067374, -1.369514, -2.578460, -0.764415, 1.570796, 1.638171],accel_mss,speed_ms,0,blend_radius_m)
    movel([0.067446, -1.369137, -2.578720, -0.764532, 1.570796, 1.638242],accel_mss,speed_ms,0,blend_radius_m)
    movel([0.067665, -1.368841, -2.578924, -0.764624, 1.570796, 1.638462],accel_mss,speed_ms,0,blend_radius_m)
    movel([0.067820, -1.368984, -2.578825, -0.764580, 1.570796, 1.638616],accel_mss,speed_ms,0,blend_radius_m)
    movel([0.067982, -1.369133, -2.578722, -0.764534, 1.570796, 1.638778],accel_mss,speed_ms,0,blend_radius_m)
    movel([0.067952, -1.369386, -2.578548, -0.764455, 1.570796, 1.638748],accel_mss,speed_ms,0,blend_radius_m)
    movel([0.067835, -1.370008, -2.578118, -0.764263, 1.570796, 1.638632],accel_mss,speed_ms,0,blend_radius_m)
    movel([0.067755, -1.370486, -2.577788, -0.764115, 1.570796, 1.638552],accel_mss,speed_ms,0,blend_radius_m)
    movel([0.067679, -1.370980, -2.577446, -0.763963, 1.570796, 1.638475],accel_mss,speed_ms,0,blend_radius_m)
    movel([0.067578, -1.371604, -2.577014, -0.763771, 1.570796, 1.638374],accel_mss,speed_ms,0,blend_radius_m)
    movel([0.067495, -1.371960, -2.576767, -0.763662, 1.570796, 1.638292],accel_mss,speed_ms,0,blend_radius_m)
    movel([0.067314, -1.372257, -2.576561, -0.763571, 1.570796, 1.638110],accel_mss,speed_ms,0,blend_radius_m)
    speed_ms = 0.003
    movel([0.067314, -1.375572, -2.578060, -0.758757, 1.570796, 1.638110],accel_mss,speed_ms,0,blend_radius_m)
    speed_ms = 0.007
    movel([0.067188, -1.375320, -2.578236, -0.758833, 1.570796, 1.637984],accel_mss,speed_ms,0,blend_radius_m)
    movel([0.067191, -1.374902, -2.578527, -0.758960, 1.570796, 1.637988],accel_mss,speed_ms,0,blend_radius_m)
    movel([0.067248, -1.374063, -2.579111, -0.759215, 1.570796, 1.638044],accel_mss,speed_ms,0,blend_radius_m)
    movel([0.067309, -1.373351, -2.579606, -0.759432, 1.570796, 1.638105],accel_mss,speed_ms,0,blend_radius_m)
    movel([0.067374, -1.372836, -2.579964, -0.759589, 1.570796, 1.638171],accel_mss,speed_ms,0,blend_radius_m)
    movel([0.067446, -1.372460, -2.580224, -0.759705, 1.570796, 1.638242],accel_mss,speed_ms,0,blend_radius_m)
    movel([0.067665, -1.372165, -2.580429, -0.759795, 1.570796, 1.638462],accel_mss,speed_ms,0,blend_radius_m)
    movel([0.067820, -1.372308, -2.580330, -0.759751, 1.570796, 1.638616],accel_mss,speed_ms,0,blend_radius_m)
    movel([0.067982, -1.372456, -2.580227, -0.759706, 1.570796, 1.638778],accel_mss,speed_ms,0,blend_radius_m)
    movel([0.067952, -1.372709, -2.580052, -0.759628, 1.570796, 1.638748],accel_mss,speed_ms,0,blend_radius_m)
    movel([0.067835, -1.373329, -2.579621, -0.759439, 1.570796, 1.638632],accel_mss,speed_ms,0,blend_radius_m)
    movel([0.067755, -1.373806, -2.579290, -0.759293, 1.570796, 1.638552],accel_mss,speed_ms,0,blend_radius_m)
    movel([0.067679, -1.374299, -2.578947, -0.759143, 1.570796, 1.638475],accel_mss,speed_ms,0,blend_radius_m)
    movel([0.067578, -1.374921, -2.578514, -0.758954, 1.570796, 1.638374],accel_mss,speed_ms,0,blend_radius_m)
    movel([0.067495, -1.375275, -2.578267, -0.758847, 1.570796, 1.638292],accel_mss,speed_ms,0,blend_radius_m)
    movel([0.067314, -1.375572, -2.578060, -0.758757, 1.570796, 1.638110],accel_mss,speed_ms,0,blend_radius_m)
    speed_ms = 0.003
    movel([0.067314, -1.362450, -2.572012, -0.777926, 1.570796, 1.638110],accel_mss,speed_ms,0,blend_radius_m)
    speed_ms = 1.000
    movel([0.067314, -1.337303, -2.559523, -0.815563, 1.570796, 1.638110],accel_mss,speed_ms,0,blend_radius_m)
    movel([0.067891, -1.337281, -2.559537, -0.815570, 1.570796, 1.638687],accel_mss,speed_ms,0,blend_radius_m)
    movel([0.067891, -1.362429, -2.572027, -0.777933, 1.570796, 1.638687],accel_mss,speed_ms,0,blend_radius_m)
    speed_ms = 0.003
    movel([0.067891, -1.372236, -2.576575, -0.763578, 1.570796, 1.638687],accel_mss,speed_ms,0,blend_radius_m)
    speed_ms = 0.007
    movel([0.068086, -1.370934, -2.577478, -0.763977, 1.570796, 1.638882],accel_mss,speed_ms,0,blend_radius_m)
    movel([0.068314, -1.369498, -2.578470, -0.764420, 1.570796, 1.639111],accel_mss,speed_ms,0,blend_radius_m)
    movel([0.068455, -1.368883, -2.578895, -0.764611, 1.570796, 1.639251],accel_mss,speed_ms,0,blend_radius_m)
    movel([0.068616, -1.368544, -2.579128, -0.764716, 1.570796, 1.639412],accel_mss,speed_ms,0,blend_radius_m)
    movel([0.068856, -1.368334, -2.579273, -0.764782, 1.570796, 1.639652],accel_mss,speed_ms,0,blend_radius_m)
    movel([0.069268, -1.367988, -2.579511, -0.764890, 1.570796, 1.640065],accel_mss,speed_ms,0,blend_radius_m)
    movel([0.069506, -1.367501, -2.579846, -0.765042, 1.570796, 1.640303],accel_mss,speed_ms,0,blend_radius_m)
    movel([0.069487, -1.367063, -2.580147, -0.765179, 1.570796, 1.640284],accel_mss,speed_ms,0,blend_radius_m)
    movel([0.069206, -1.366852, -2.580292, -0.765245, 1.570796, 1.640003],accel_mss,speed_ms,0,blend_radius_m)
    movel([0.068881, -1.366852, -2.580292, -0.765245, 1.570796, 1.639677],accel_mss,speed_ms,0,blend_radius_m)
    movel([0.068537, -1.367087, -2.580131, -0.765171, 1.570796, 1.639333],accel_mss,speed_ms,0,blend_radius_m)
    movel([0.068259, -1.367393, -2.579920, -0.765076, 1.570796, 1.639055],accel_mss,speed_ms,0,blend_radius_m)
    movel([0.068159, -1.367743, -2.579680, -0.764966, 1.570796, 1.638956],accel_mss,speed_ms,0,blend_radius_m)
    movel([0.068095, -1.368023, -2.579487, -0.764879, 1.570796, 1.638891],accel_mss,speed_ms,0,blend_radius_m)
    movel([0.067951, -1.368268, -2.579319, -0.764803, 1.570796, 1.638748],accel_mss,speed_ms,0,blend_radius_m)
    movel([0.067551, -1.368495, -2.579162, -0.764732, 1.570796, 1.638348],accel_mss,speed_ms,0,blend_radius_m)
    movel([0.067363, -1.368371, -2.579248, -0.764770, 1.570796, 1.638159],accel_mss,speed_ms,0,blend_radius_m)
    movel([0.067160, -1.368082, -2.579447, -0.764860, 1.570796, 1.637956],accel_mss,speed_ms,0,blend_radius_m)
    movel([0.066968, -1.367808, -2.579635, -0.764946, 1.570796, 1.637764],accel_mss,speed_ms,0,blend_radius_m)
    movel([0.066743, -1.367664, -2.579734, -0.764991, 1.570796, 1.637539],accel_mss,speed_ms,0,blend_radius_m)
    movel([0.066454, -1.367638, -2.579752, -0.764999, 1.570796, 1.637251],accel_mss,speed_ms,0,blend_radius_m)
    movel([0.066073, -1.367717, -2.579698, -0.764974, 1.570796, 1.636869],accel_mss,speed_ms,0,blend_radius_m)
    movel([0.065765, -1.367878, -2.579587, -0.764924, 1.570796, 1.636562],accel_mss,speed_ms,0,blend_radius_m)
    movel([0.065486, -1.368148, -2.579401, -0.764840, 1.570796, 1.636282],accel_mss,speed_ms,0,blend_radius_m)
    movel([0.065298, -1.368462, -2.579185, -0.764742, 1.570796, 1.636095],accel_mss,speed_ms,0,blend_radius_m)
    movel([0.065249, -1.368750, -2.578987, -0.764653, 1.570796, 1.636045],accel_mss,speed_ms,0,blend_radius_m)
    movel([0.065355, -1.368924, -2.578866, -0.764598, 1.570796, 1.636151],accel_mss,speed_ms,0,blend_radius_m)
    movel([0.065666, -1.369073, -2.578764, -0.764552, 1.570796, 1.636462],accel_mss,speed_ms,0,blend_radius_m)
    movel([0.066034, -1.369155, -2.578708, -0.764527, 1.570796, 1.636830],accel_mss,speed_ms,0,blend_radius_m)
    movel([0.066342, -1.369120, -2.578732, -0.764538, 1.570796, 1.637138],accel_mss,speed_ms,0,blend_radius_m)
    movel([0.066688, -1.369137, -2.578720, -0.764532, 1.570796, 1.637484],accel_mss,speed_ms,0,blend_radius_m)
    movel([0.066870, -1.369408, -2.578532, -0.764448, 1.570796, 1.637666],accel_mss,speed_ms,0,blend_radius_m)
    movel([0.066903, -1.370060, -2.578083, -0.764247, 1.570796, 1.637699],accel_mss,speed_ms,0,blend_radius_m)
    movel([0.066779, -1.371453, -2.577118, -0.763817, 1.570796, 1.637575],accel_mss,speed_ms,0,blend_radius_m)
    movel([0.066708, -1.372078, -2.576685, -0.763626, 1.570796, 1.637504],accel_mss,speed_ms,0,blend_radius_m)
    movel([0.066649, -1.372354, -2.576493, -0.763541, 1.570796, 1.637446],accel_mss,speed_ms,0,blend_radius_m)
    movel([0.066450, -1.372560, -2.576351, -0.763479, 1.570796, 1.637247],accel_mss,speed_ms,0,blend_radius_m)
    movel([0.066231, -1.372466, -2.576416, -0.763507, 1.570796, 1.637027],accel_mss,speed_ms,0,blend_radius_m)
    movel([0.066132, -1.372239, -2.576573, -0.763577, 1.570796, 1.636928],accel_mss,speed_ms,0,blend_radius_m)
    movel([0.065933, -1.372130, -2.576649, -0.763610, 1.570796, 1.636729],accel_mss,speed_ms,0,blend_radius_m)
    movel([0.065974, -1.371889, -2.576816, -0.763684, 1.570796, 1.636770],accel_mss,speed_ms,0,blend_radius_m)
    movel([0.065993, -1.371608, -2.577011, -0.763770, 1.570796, 1.636789],accel_mss,speed_ms,0,blend_radius_m)
    movel([0.065755, -1.371549, -2.577052, -0.763788, 1.570796, 1.636552],accel_mss,speed_ms,0,blend_radius_m)
    movel([0.065388, -1.371592, -2.577022, -0.763775, 1.570796, 1.636185],accel_mss,speed_ms,0,blend_radius_m)
    movel([0.064410, -1.371541, -2.577057, -0.763790, 1.570796, 1.635206],accel_mss,speed_ms,0,blend_radius_m)
    movel([0.063662, -1.371220, -2.577280, -0.763889, 1.570796, 1.634458],accel_mss,speed_ms,0,blend_radius_m)
    movel([0.063073, -1.370714, -2.577630, -0.764045, 1.570796, 1.633869],accel_mss,speed_ms,0,blend_radius_m)
    movel([0.062754, -1.370096, -2.578057, -0.764235, 1.570796, 1.633550],accel_mss,speed_ms,0,blend_radius_m)
    movel([0.062718, -1.369302, -2.578606, -0.764481, 1.570796, 1.633515],accel_mss,speed_ms,0,blend_radius_m)
    movel([0.062983, -1.368306, -2.579293, -0.764791, 1.570796, 1.633779],accel_mss,speed_ms,0,blend_radius_m)
    movel([0.063493, -1.367264, -2.580009, -0.765116, 1.570796, 1.634289],accel_mss,speed_ms,0,blend_radius_m)
    movel([0.064187, -1.366327, -2.580653, -0.765410, 1.570796, 1.634984],accel_mss,speed_ms,0,blend_radius_m)
    movel([0.064468, -1.366042, -2.580848, -0.765499, 1.570796, 1.635264],accel_mss,speed_ms,0,blend_radius_m)
    movel([0.064844, -1.365705, -2.581079, -0.765605, 1.570796, 1.635641],accel_mss,speed_ms,0,blend_radius_m)
    movel([0.065259, -1.365367, -2.581310, -0.765712, 1.570796, 1.636055],accel_mss,speed_ms,0,blend_radius_m)
    movel([0.065655, -1.365077, -2.581508, -0.765803, 1.570796, 1.636451],accel_mss,speed_ms,0,blend_radius_m)
    movel([0.066240, -1.364690, -2.581773, -0.765926, 1.570796, 1.637037],accel_mss,speed_ms,0,blend_radius_m)
    movel([0.066630, -1.364481, -2.581916, -0.765992, 1.570796, 1.637427],accel_mss,speed_ms,0,blend_radius_m)
    movel([0.067072, -1.364316, -2.582029, -0.766044, 1.570796, 1.637868],accel_mss,speed_ms,0,blend_radius_m)
    movel([0.067932, -1.364064, -2.582200, -0.766124, 1.570796, 1.638728],accel_mss,speed_ms,0,blend_radius_m)
    movel([0.068629, -1.363881, -2.582325, -0.766182, 1.570796, 1.639426],accel_mss,speed_ms,0,blend_radius_m)
    movel([0.069134, -1.363776, -2.582397, -0.766216, 1.570796, 1.639930],accel_mss,speed_ms,0,blend_radius_m)
    movel([0.069542, -1.363727, -2.582430, -0.766231, 1.570796, 1.640338],accel_mss,speed_ms,0,blend_radius_m)
    movel([0.069913, -1.363729, -2.582429, -0.766231, 1.570796, 1.640709],accel_mss,speed_ms,0,blend_radius_m)
    movel([0.070682, -1.363828, -2.582362, -0.766199, 1.570796, 1.641478],accel_mss,speed_ms,0,blend_radius_m)
    movel([0.071270, -1.364006, -2.582240, -0.766143, 1.570796, 1.642066],accel_mss,speed_ms,0,blend_radius_m)
    movel([0.071742, -1.364286, -2.582049, -0.766054, 1.570796, 1.642538],accel_mss,speed_ms,0,blend_radius_m)
    movel([0.072153, -1.364697, -2.581768, -0.765924, 1.570796, 1.642949],accel_mss,speed_ms,0,blend_radius_m)
    movel([0.072432, -1.365078, -2.581508, -0.765803, 1.570796, 1.643228],accel_mss,speed_ms,0,blend_radius_m)
    movel([0.072562, -1.365356, -2.581318, -0.765716, 1.570796, 1.643358],accel_mss,speed_ms,0,blend_radius_m)
    movel([0.072615, -1.365695, -2.581085, -0.765608, 1.570796, 1.643412],accel_mss,speed_ms,0,blend_radius_m)
    movel([0.072625, -1.366311, -2.580663, -0.765415, 1.570796, 1.643422],accel_mss,speed_ms,0,blend_radius_m)
    movel([0.072624, -1.366703, -2.580394, -0.765292, 1.570796, 1.643421],accel_mss,speed_ms,0,blend_radius_m)
    movel([0.072626, -1.367039, -2.580163, -0.765186, 1.570796, 1.643422],accel_mss,speed_ms,0,blend_radius_m)
    movel([0.072628, -1.367330, -2.579964, -0.765095, 1.570796, 1.643425],accel_mss,speed_ms,0,blend_radius_m)
    movel([0.072329, -1.367646, -2.579746, -0.764996, 1.570796, 1.643125],accel_mss,speed_ms,0,blend_radius_m)
    movel([0.072081, -1.368084, -2.579445, -0.764860, 1.570796, 1.642878],accel_mss,speed_ms,0,blend_radius_m)
    movel([0.071908, -1.368353, -2.579260, -0.764776, 1.570796, 1.642704],accel_mss,speed_ms,0,blend_radius_m)
    movel([0.071728, -1.368608, -2.579084, -0.764697, 1.570796, 1.642524],accel_mss,speed_ms,0,blend_radius_m)
    movel([0.071129, -1.369231, -2.578655, -0.764503, 1.570796, 1.641925],accel_mss,speed_ms,0,blend_radius_m)
    movel([0.070532, -1.369679, -2.578346, -0.764364, 1.570796, 1.641329],accel_mss,speed_ms,0,blend_radius_m)
    movel([0.069917, -1.370062, -2.578081, -0.764246, 1.570796, 1.640713],accel_mss,speed_ms,0,blend_radius_m)
    movel([0.069427, -1.370278, -2.577932, -0.764179, 1.570796, 1.640223],accel_mss,speed_ms,0,blend_radius_m)
    movel([0.069053, -1.370439, -2.577821, -0.764130, 1.570796, 1.639849],accel_mss,speed_ms,0,blend_radius_m)
    movel([0.068800, -1.370627, -2.577690, -0.764071, 1.570796, 1.639597],accel_mss,speed_ms,0,blend_radius_m)
    movel([0.068643, -1.370899, -2.577502, -0.763988, 1.570796, 1.639439],accel_mss,speed_ms,0,blend_radius_m)
    movel([0.068529, -1.371298, -2.577226, -0.763865, 1.570796, 1.639325],accel_mss,speed_ms,0,blend_radius_m)
    movel([0.068476, -1.371655, -2.576978, -0.763755, 1.570796, 1.639272],accel_mss,speed_ms,0,blend_radius_m)
    movel([0.068694, -1.371767, -2.576901, -0.763721, 1.570796, 1.639490],accel_mss,speed_ms,0,blend_radius_m)
    movel([0.068466, -1.372049, -2.576705, -0.763635, 1.570796, 1.639263],accel_mss,speed_ms,0,blend_radius_m)
    movel([0.067891, -1.372236, -2.576575, -0.763578, 1.570796, 1.638687],accel_mss,speed_ms,0,blend_radius_m)
    speed_ms = 0.003
    movel([0.067891, -1.375551, -2.578075, -0.758763, 1.570796, 1.638687],accel_mss,speed_ms,0,blend_radius_m)
    speed_ms = 0.007
    movel([0.068086, -1.374253, -2.578979, -0.759157, 1.570796, 1.638882],accel_mss,speed_ms,0,blend_radius_m)
    movel([0.068314, -1.372821, -2.579974, -0.759594, 1.570796, 1.639111],accel_mss,speed_ms,0,blend_radius_m)
    movel([0.068455, -1.372207, -2.580399, -0.759782, 1.570796, 1.639251],accel_mss,speed_ms,0,blend_radius_m)
    movel([0.068616, -1.371869, -2.580634, -0.759886, 1.570796, 1.639412],accel_mss,speed_ms,0,blend_radius_m)
    movel([0.068856, -1.371659, -2.580779, -0.759951, 1.570796, 1.639652],accel_mss,speed_ms,0,blend_radius_m)
    movel([0.069268, -1.371315, -2.581018, -0.760057, 1.570796, 1.640065],accel_mss,speed_ms,0,blend_radius_m)
    movel([0.069506, -1.370829, -2.581353, -0.760207, 1.570796, 1.640303],accel_mss,speed_ms,0,blend_radius_m)
    movel([0.069487, -1.370391, -2.581655, -0.760342, 1.570796, 1.640284],accel_mss,speed_ms,0,blend_radius_m)
    movel([0.069206, -1.370181, -2.581800, -0.760407, 1.570796, 1.640003],accel_mss,speed_ms,0,blend_radius_m)
    movel([0.068881, -1.370181, -2.581801, -0.760407, 1.570796, 1.639677],accel_mss,speed_ms,0,blend_radius_m)
    movel([0.068537, -1.370416, -2.581639, -0.760335, 1.570796, 1.639333],accel_mss,speed_ms,0,blend_radius_m)
    movel([0.068259, -1.370721, -2.581428, -0.760240, 1.570796, 1.639055],accel_mss,speed_ms,0,blend_radius_m)
    movel([0.068159, -1.371070, -2.581186, -0.760132, 1.570796, 1.638956],accel_mss,speed_ms,0,blend_radius_m)
    movel([0.068095, -1.371349, -2.580994, -0.760046, 1.570796, 1.638891],accel_mss,speed_ms,0,blend_radius_m)
    movel([0.067951, -1.371593, -2.580825, -0.759971, 1.570796, 1.638748],accel_mss,speed_ms,0,blend_radius_m)
    movel([0.067551, -1.371820, -2.580668, -0.759901, 1.570796, 1.638348],accel_mss,speed_ms,0,blend_radius_m)
    movel([0.067363, -1.371696, -2.580753, -0.759939, 1.570796, 1.638159],accel_mss,speed_ms,0,blend_radius_m)
    movel([0.067160, -1.371408, -2.580953, -0.760028, 1.570796, 1.637956],accel_mss,speed_ms,0,blend_radius_m)
    movel([0.066968, -1.371135, -2.581142, -0.760112, 1.570796, 1.637764],accel_mss,speed_ms,0,blend_radius_m)
    movel([0.066743, -1.370991, -2.581241, -0.760157, 1.570796, 1.637539],accel_mss,speed_ms,0,blend_radius_m)
    movel([0.066454, -1.370965, -2.581259, -0.760165, 1.570796, 1.637251],accel_mss,speed_ms,0,blend_radius_m)
    movel([0.066073, -1.371044, -2.581205, -0.760140, 1.570796, 1.636869],accel_mss,speed_ms,0,blend_radius_m)
    movel([0.065765, -1.371204, -2.581094, -0.760091, 1.570796, 1.636562],accel_mss,speed_ms,0,blend_radius_m)
    movel([0.065486, -1.371474, -2.580907, -0.760008, 1.570796, 1.636282],accel_mss,speed_ms,0,blend_radius_m)
    movel([0.065298, -1.371787, -2.580690, -0.759911, 1.570796, 1.636095],accel_mss,speed_ms,0,blend_radius_m)
    movel([0.065249, -1.372074, -2.580492, -0.759823, 1.570796, 1.636045],accel_mss,speed_ms,0,blend_radius_m)
    movel([0.065355, -1.372248, -2.580371, -0.759770, 1.570796, 1.636151],accel_mss,speed_ms,0,blend_radius_m)
    movel([0.065666, -1.372396, -2.580268, -0.759724, 1.570796, 1.636462],accel_mss,speed_ms,0,blend_radius_m)
    movel([0.066034, -1.372478, -2.580212, -0.759699, 1.570796, 1.636830],accel_mss,speed_ms,0,blend_radius_m)
    movel([0.066342, -1.372443, -2.580236, -0.759710, 1.570796, 1.637138],accel_mss,speed_ms,0,blend_radius_m)
    movel([0.066688, -1.372460, -2.580224, -0.759705, 1.570796, 1.637484],accel_mss,speed_ms,0,blend_radius_m)
    movel([0.066870, -1.372731, -2.580036, -0.759622, 1.570796, 1.637666],accel_mss,speed_ms,0,blend_radius_m)
    movel([0.066903, -1.373380, -2.579586, -0.759423, 1.570796, 1.637699],accel_mss,speed_ms,0,blend_radius_m)
    movel([0.066779, -1.374771, -2.578619, -0.759000, 1.570796, 1.637575],accel_mss,speed_ms,0,blend_radius_m)
    movel([0.066708, -1.375394, -2.578185, -0.758811, 1.570796, 1.637504],accel_mss,speed_ms,0,blend_radius_m)
    movel([0.066649, -1.375669, -2.577992, -0.758728, 1.570796, 1.637446],accel_mss,speed_ms,0,blend_radius_m)
    movel([0.066450, -1.375874, -2.577849, -0.758666, 1.570796, 1.637247],accel_mss,speed_ms,0,blend_radius_m)
    movel([0.066231, -1.375780, -2.577915, -0.758694, 1.570796, 1.637027],accel_mss,speed_ms,0,blend_radius_m)
    movel([0.066132, -1.375554, -2.578073, -0.758762, 1.570796, 1.636928],accel_mss,speed_ms,0,blend_radius_m)
    movel([0.065933, -1.375445, -2.578149, -0.758795, 1.570796, 1.636729],accel_mss,speed_ms,0,blend_radius_m)
    movel([0.065974, -1.375205, -2.578316, -0.758868, 1.570796, 1.636770],accel_mss,speed_ms,0,blend_radius_m)
    movel([0.065993, -1.374925, -2.578511, -0.758953, 1.570796, 1.636789],accel_mss,speed_ms,0,blend_radius_m)
    movel([0.065755, -1.374866, -2.578552, -0.758971, 1.570796, 1.636552],accel_mss,speed_ms,0,blend_radius_m)
    movel([0.065388, -1.374909, -2.578523, -0.758958, 1.570796, 1.636185],accel_mss,speed_ms,0,blend_radius_m)
    movel([0.064410, -1.374858, -2.578558, -0.758973, 1.570796, 1.635206],accel_mss,speed_ms,0,blend_radius_m)
    movel([0.063662, -1.374538, -2.578781, -0.759070, 1.570796, 1.634458],accel_mss,speed_ms,0,blend_radius_m)
    movel([0.063073, -1.374033, -2.579132, -0.759224, 1.570796, 1.633869],accel_mss,speed_ms,0,blend_radius_m)
    movel([0.062754, -1.373417, -2.579560, -0.759412, 1.570796, 1.633550],accel_mss,speed_ms,0,blend_radius_m)
    movel([0.062718, -1.372625, -2.580110, -0.759654, 1.570796, 1.633515],accel_mss,speed_ms,0,blend_radius_m)
    movel([0.062983, -1.371631, -2.580799, -0.759959, 1.570796, 1.633779],accel_mss,speed_ms,0,blend_radius_m)
    movel([0.063493, -1.370592, -2.581517, -0.760280, 1.570796, 1.634289],accel_mss,speed_ms,0,blend_radius_m)
    movel([0.064187, -1.369657, -2.582162, -0.760570, 1.570796, 1.634984],accel_mss,speed_ms,0,blend_radius_m)
    movel([0.064468, -1.369373, -2.582357, -0.760658, 1.570796, 1.635264],accel_mss,speed_ms,0,blend_radius_m)
    movel([0.064844, -1.369037, -2.582589, -0.760763, 1.570796, 1.635641],accel_mss,speed_ms,0,blend_radius_m)
    movel([0.065259, -1.368700, -2.582821, -0.760868, 1.570796, 1.636055],accel_mss,speed_ms,0,blend_radius_m)
    movel([0.065655, -1.368412, -2.583019, -0.760958, 1.570796, 1.636451],accel_mss,speed_ms,0,blend_radius_m)
    movel([0.066240, -1.368025, -2.583285, -0.761079, 1.570796, 1.637037],accel_mss,speed_ms,0,blend_radius_m)
    movel([0.066630, -1.367817, -2.583428, -0.761144, 1.570796, 1.637427],accel_mss,speed_ms,0,blend_radius_m)
    movel([0.067072, -1.367652, -2.583541, -0.761196, 1.570796, 1.637868],accel_mss,speed_ms,0,blend_radius_m)
    movel([0.067932, -1.367401, -2.583713, -0.761275, 1.570796, 1.638728],accel_mss,speed_ms,0,blend_radius_m)
    movel([0.068629, -1.367218, -2.583839, -0.761332, 1.570796, 1.639426],accel_mss,speed_ms,0,blend_radius_m)
    movel([0.069134, -1.367114, -2.583910, -0.761365, 1.570796, 1.639930],accel_mss,speed_ms,0,blend_radius_m)
    movel([0.069542, -1.367065, -2.583944, -0.761380, 1.570796, 1.640338],accel_mss,speed_ms,0,blend_radius_m)
    movel([0.069913, -1.367066, -2.583943, -0.761380, 1.570796, 1.640709],accel_mss,speed_ms,0,blend_radius_m)
    movel([0.070682, -1.367165, -2.583875, -0.761349, 1.570796, 1.641478],accel_mss,speed_ms,0,blend_radius_m)
    movel([0.071270, -1.367343, -2.583753, -0.761293, 1.570796, 1.642066],accel_mss,speed_ms,0,blend_radius_m)
    movel([0.071742, -1.367622, -2.583561, -0.761205, 1.570796, 1.642538],accel_mss,speed_ms,0,blend_radius_m)
    movel([0.072153, -1.368032, -2.583280, -0.761077, 1.570796, 1.642949],accel_mss,speed_ms,0,blend_radius_m)
    movel([0.072432, -1.368412, -2.583019, -0.760958, 1.570796, 1.643228],accel_mss,speed_ms,0,blend_radius_m)
    movel([0.072562, -1.368689, -2.582828, -0.760872, 1.570796, 1.643358],accel_mss,speed_ms,0,blend_radius_m)
    movel([0.072615, -1.369028, -2.582595, -0.760766, 1.570796, 1.643412],accel_mss,speed_ms,0,blend_radius_m)
    movel([0.072625, -1.369642, -2.582173, -0.760575, 1.570796, 1.643422],accel_mss,speed_ms,0,blend_radius_m)
    movel([0.072624, -1.370033, -2.581903, -0.760453, 1.570796, 1.643421],accel_mss,speed_ms,0,blend_radius_m)
    movel([0.072626, -1.370368, -2.581671, -0.760349, 1.570796, 1.643422],accel_mss,speed_ms,0,blend_radius_m)
    movel([0.072628, -1.370658, -2.581471, -0.760260, 1.570796, 1.643425],accel_mss,speed_ms,0,blend_radius_m)
    movel([0.072329, -1.370973, -2.581253, -0.760162, 1.570796, 1.643125],accel_mss,speed_ms,0,blend_radius_m)
    movel([0.072081, -1.371410, -2.580951, -0.760027, 1.570796, 1.642878],accel_mss,speed_ms,0,blend_radius_m)
    movel([0.071908, -1.371678, -2.580766, -0.759945, 1.570796, 1.642704],accel_mss,speed_ms,0,blend_radius_m)
    movel([0.071728, -1.371933, -2.580590, -0.759867, 1.570796, 1.642524],accel_mss,speed_ms,0,blend_radius_m)
    movel([0.071129, -1.372554, -2.580159, -0.759676, 1.570796, 1.641925],accel_mss,speed_ms,0,blend_radius_m)
    movel([0.070532, -1.373001, -2.579849, -0.759539, 1.570796, 1.641329],accel_mss,speed_ms,0,blend_radius_m)
    movel([0.069917, -1.373383, -2.579584, -0.759422, 1.570796, 1.640713],accel_mss,speed_ms,0,blend_radius_m)
    movel([0.069427, -1.373598, -2.579434, -0.759356, 1.570796, 1.640223],accel_mss,speed_ms,0,blend_radius_m)
    movel([0.069053, -1.373758, -2.579323, -0.759308, 1.570796, 1.639849],accel_mss,speed_ms,0,blend_radius_m)
    movel([0.068800, -1.373947, -2.579192, -0.759250, 1.570796, 1.639597],accel_mss,speed_ms,0,blend_radius_m)
    movel([0.068643, -1.374217, -2.579004, -0.759168, 1.570796, 1.639439],accel_mss,speed_ms,0,blend_radius_m)
    movel([0.068529, -1.374615, -2.578727, -0.759047, 1.570796, 1.639325],accel_mss,speed_ms,0,blend_radius_m)
    movel([0.068476, -1.374972, -2.578479, -0.758939, 1.570796, 1.639272],accel_mss,speed_ms,0,blend_radius_m)
    movel([0.068694, -1.375083, -2.578401, -0.758905, 1.570796, 1.639490],accel_mss,speed_ms,0,blend_radius_m)
    movel([0.068466, -1.375365, -2.578205, -0.758820, 1.570796, 1.639263],accel_mss,speed_ms,0,blend_radius_m)
    movel([0.067891, -1.375551, -2.578075, -0.758763, 1.570796, 1.638687],accel_mss,speed_ms,0,blend_radius_m)
    speed_ms = 0.003
    movel([0.067891, -1.362429, -2.572027, -0.777933, 1.570796, 1.638687],accel_mss,speed_ms,0,blend_radius_m)
    speed_ms = 1.000
    movel([0.067891, -1.337281, -2.559537, -0.815570, 1.570796, 1.638687],accel_mss,speed_ms,0,blend_radius_m)
    movel([0.068557, -1.332885, -2.562423, -0.817081, 1.570796, 1.639354],accel_mss,speed_ms,0,blend_radius_m)
    movel([0.068557, -1.358109, -2.574969, -0.779311, 1.570796, 1.639354],accel_mss,speed_ms,0,blend_radius_m)
    speed_ms = 0.003
    movel([0.068557, -1.367949, -2.579538, -0.764902, 1.570796, 1.639354],accel_mss,speed_ms,0,blend_radius_m)
    speed_ms = 0.007
    movel([0.068577, -1.367549, -2.579813, -0.765027, 1.570796, 1.639373],accel_mss,speed_ms,0,blend_radius_m)
    movel([0.068828, -1.367296, -2.579987, -0.765106, 1.570796, 1.639624],accel_mss,speed_ms,0,blend_radius_m)
    movel([0.069143, -1.367298, -2.579986, -0.765105, 1.570796, 1.639939],accel_mss,speed_ms,0,blend_radius_m)
    movel([0.069072, -1.367533, -2.579824, -0.765032, 1.570796, 1.639868],accel_mss,speed_ms,0,blend_radius_m)
    movel([0.068842, -1.367743, -2.579680, -0.764966, 1.570796, 1.639638],accel_mss,speed_ms,0,blend_radius_m)
    movel([0.068557, -1.367949, -2.579538, -0.764902, 1.570796, 1.639354],accel_mss,speed_ms,0,blend_radius_m)
    speed_ms = 0.003
    movel([0.068557, -1.371275, -2.581045, -0.760069, 1.570796, 1.639354],accel_mss,speed_ms,0,blend_radius_m)
    speed_ms = 0.007
    movel([0.068577, -1.370876, -2.581320, -0.760192, 1.570796, 1.639373],accel_mss,speed_ms,0,blend_radius_m)
    movel([0.068828, -1.370624, -2.581495, -0.760270, 1.570796, 1.639624],accel_mss,speed_ms,0,blend_radius_m)
    movel([0.069143, -1.370626, -2.581493, -0.760270, 1.570796, 1.639939],accel_mss,speed_ms,0,blend_radius_m)
    movel([0.069072, -1.370860, -2.581332, -0.760197, 1.570796, 1.639868],accel_mss,speed_ms,0,blend_radius_m)
    movel([0.068842, -1.371070, -2.581187, -0.760132, 1.570796, 1.639638],accel_mss,speed_ms,0,blend_radius_m)
    movel([0.068557, -1.371275, -2.581045, -0.760069, 1.570796, 1.639354],accel_mss,speed_ms,0,blend_radius_m)
    speed_ms = 0.003
    movel([0.068557, -1.358109, -2.574969, -0.779311, 1.570796, 1.639354],accel_mss,speed_ms,0,blend_radius_m)
    speed_ms = 1.000
    movel([0.068557, -1.332885, -2.562423, -0.817081, 1.570796, 1.639354],accel_mss,speed_ms,0,blend_radius_m)
    movel([0.066722, -1.333449, -2.562054, -0.816886, 1.570796, 1.637519],accel_mss,speed_ms,0,blend_radius_m)
    movel([0.066722, -1.358664, -2.574592, -0.779133, 1.570796, 1.637519],accel_mss,speed_ms,0,blend_radius_m)
    speed_ms = 0.003
    movel([0.066722, -1.368499, -2.579159, -0.764730, 1.570796, 1.637519],accel_mss,speed_ms,0,blend_radius_m)
    speed_ms = 0.007
    movel([0.066563, -1.368732, -2.578999, -0.764658, 1.570796, 1.637359],accel_mss,speed_ms,0,blend_radius_m)
    movel([0.066206, -1.368695, -2.579024, -0.764669, 1.570796, 1.637002],accel_mss,speed_ms,0,blend_radius_m)
    movel([0.065869, -1.368561, -2.579117, -0.764711, 1.570796, 1.636665],accel_mss,speed_ms,0,blend_radius_m)
    movel([0.065944, -1.368236, -2.579341, -0.764812, 1.570796, 1.636740],accel_mss,speed_ms,0,blend_radius_m)
    movel([0.066166, -1.368019, -2.579490, -0.764880, 1.570796, 1.636963],accel_mss,speed_ms,0,blend_radius_m)
    movel([0.066451, -1.368162, -2.579392, -0.764836, 1.570796, 1.637247],accel_mss,speed_ms,0,blend_radius_m)
    movel([0.066639, -1.368330, -2.579276, -0.764783, 1.570796, 1.637435],accel_mss,speed_ms,0,blend_radius_m)
    speed_ms = 0.003
    movel([0.066722, -1.371824, -2.580665, -0.759900, 1.570796, 1.637519],accel_mss,speed_ms,0,blend_radius_m)
    speed_ms = 0.007
    movel([0.066563, -1.372056, -2.580504, -0.759829, 1.570796, 1.637359],accel_mss,speed_ms,0,blend_radius_m)
    movel([0.066206, -1.372020, -2.580529, -0.759840, 1.570796, 1.637002],accel_mss,speed_ms,0,blend_radius_m)
    movel([0.065869, -1.371886, -2.580622, -0.759881, 1.570796, 1.636665],accel_mss,speed_ms,0,blend_radius_m)
    movel([0.065944, -1.371562, -2.580847, -0.759981, 1.570796, 1.636740],accel_mss,speed_ms,0,blend_radius_m)
    movel([0.066166, -1.371346, -2.580996, -0.760047, 1.570796, 1.636963],accel_mss,speed_ms,0,blend_radius_m)
    movel([0.066451, -1.371488, -2.580898, -0.760004, 1.570796, 1.637247],accel_mss,speed_ms,0,blend_radius_m)
    movel([0.066639, -1.371655, -2.580782, -0.759952, 1.570796, 1.637435],accel_mss,speed_ms,0,blend_radius_m)
    speed_ms = 0.003
    movel([0.066722, -1.358664, -2.574592, -0.779133, 1.570796, 1.637519],accel_mss,speed_ms,0,blend_radius_m)
    speed_ms = 1.000
    movel([0.066722, -1.333449, -2.562054, -0.816886, 1.570796, 1.637519],accel_mss,speed_ms,0,blend_radius_m)
    movel([0.065746, -1.318776, -2.571512, -0.822101, 1.570796, 1.636542],accel_mss,speed_ms,0,blend_radius_m)
    movel([0.065746, -1.344239, -2.584239, -0.783911, 1.570796, 1.636542],accel_mss,speed_ms,0,blend_radius_m)
    speed_ms = 0.003
    movel([0.065746, -1.354182, -2.588877, -0.769330, 1.570796, 1.636542],accel_mss,speed_ms,0,blend_radius_m)
    speed_ms = 0.007
    movel([0.065772, -1.353710, -2.589193, -0.769486, 1.570796, 1.636568],accel_mss,speed_ms,0,blend_radius_m)
    movel([0.066112, -1.352862, -2.589759, -0.769768, 1.570796, 1.636908],accel_mss,speed_ms,0,blend_radius_m)
    movel([0.067083, -1.350617, -2.591252, -0.770519, 1.570796, 1.637880],accel_mss,speed_ms,0,blend_radius_m)
    movel([0.067719, -1.349136, -2.592234, -0.771019, 1.570796, 1.638515],accel_mss,speed_ms,0,blend_radius_m)
    movel([0.068073, -1.348257, -2.592815, -0.771317, 1.570796, 1.638869],accel_mss,speed_ms,0,blend_radius_m)
    movel([0.068273, -1.347685, -2.593193, -0.771511, 1.570796, 1.639069],accel_mss,speed_ms,0,blend_radius_m)
    movel([0.068106, -1.347511, -2.593307, -0.771570, 1.570796, 1.638903],accel_mss,speed_ms,0,blend_radius_m)
    movel([0.067773, -1.347577, -2.593264, -0.771548, 1.570796, 1.638570],accel_mss,speed_ms,0,blend_radius_m)
    movel([0.067262, -1.347717, -2.593172, -0.771501, 1.570796, 1.638058],accel_mss,speed_ms,0,blend_radius_m)
    movel([0.066457, -1.347971, -2.593004, -0.771414, 1.570796, 1.637253],accel_mss,speed_ms,0,blend_radius_m)
    movel([0.065785, -1.348180, -2.592866, -0.771343, 1.570796, 1.636581],accel_mss,speed_ms,0,blend_radius_m)
    movel([0.065232, -1.348336, -2.592763, -0.771290, 1.570796, 1.636028],accel_mss,speed_ms,0,blend_radius_m)
    movel([0.064791, -1.348447, -2.592690, -0.771252, 1.570796, 1.635588],accel_mss,speed_ms,0,blend_radius_m)
    movel([0.064973, -1.347487, -2.593324, -0.771579, 1.570796, 1.635770],accel_mss,speed_ms,0,blend_radius_m)
    movel([0.065442, -1.346342, -2.594078, -0.771970, 1.570796, 1.636238],accel_mss,speed_ms,0,blend_radius_m)
    movel([0.066182, -1.344629, -2.595202, -0.772557, 1.570796, 1.636979],accel_mss,speed_ms,0,blend_radius_m)
    movel([0.066820, -1.343178, -2.596152, -0.773059, 1.570796, 1.637617],accel_mss,speed_ms,0,blend_radius_m)
    movel([0.067378, -1.341927, -2.596969, -0.773494, 1.570796, 1.638175],accel_mss,speed_ms,0,blend_radius_m)
    movel([0.067871, -1.340832, -2.597682, -0.773876, 1.570796, 1.638668],accel_mss,speed_ms,0,blend_radius_m)
    movel([0.068273, -1.340444, -2.597934, -0.774011, 1.570796, 1.639070],accel_mss,speed_ms,0,blend_radius_m)
    movel([0.070568, -1.339691, -2.598423, -0.774275, 1.570796, 1.641364],accel_mss,speed_ms,0,blend_radius_m)
    movel([0.072875, -1.338962, -2.598895, -0.774532, 1.570796, 1.643671],accel_mss,speed_ms,0,blend_radius_m)
    movel([0.073115, -1.339033, -2.598849, -0.774507, 1.570796, 1.643911],accel_mss,speed_ms,0,blend_radius_m)
    movel([0.072689, -1.339919, -2.598275, -0.774195, 1.570796, 1.643486],accel_mss,speed_ms,0,blend_radius_m)
    movel([0.072189, -1.340820, -2.597690, -0.773880, 1.570796, 1.642986],accel_mss,speed_ms,0,blend_radius_m)
    movel([0.071589, -1.341857, -2.597014, -0.773518, 1.570796, 1.642385],accel_mss,speed_ms,0,blend_radius_m)
    movel([0.070780, -1.343250, -2.596105, -0.773034, 1.570796, 1.641576],accel_mss,speed_ms,0,blend_radius_m)
    movel([0.070360, -1.344020, -2.595601, -0.772768, 1.570796, 1.641156],accel_mss,speed_ms,0,blend_radius_m)
    movel([0.070135, -1.344497, -2.595289, -0.772603, 1.570796, 1.640931],accel_mss,speed_ms,0,blend_radius_m)
    movel([0.070293, -1.344677, -2.595171, -0.772541, 1.570796, 1.641090],accel_mss,speed_ms,0,blend_radius_m)
    movel([0.070585, -1.344629, -2.595202, -0.772558, 1.570796, 1.641381],accel_mss,speed_ms,0,blend_radius_m)
    movel([0.071041, -1.344508, -2.595281, -0.772599, 1.570796, 1.641837],accel_mss,speed_ms,0,blend_radius_m)
    movel([0.071762, -1.344282, -2.595430, -0.772677, 1.570796, 1.642559],accel_mss,speed_ms,0,blend_radius_m)
    movel([0.072728, -1.343981, -2.595627, -0.772781, 1.570796, 1.643524],accel_mss,speed_ms,0,blend_radius_m)
    movel([0.073151, -1.343887, -2.595689, -0.772814, 1.570796, 1.643947],accel_mss,speed_ms,0,blend_radius_m)
    movel([0.073323, -1.344073, -2.595566, -0.772749, 1.570796, 1.644120],accel_mss,speed_ms,0,blend_radius_m)
    movel([0.072183, -1.345650, -2.594532, -0.772207, 1.570796, 1.642979],accel_mss,speed_ms,0,blend_radius_m)
    movel([0.070974, -1.347290, -2.593453, -0.771646, 1.570796, 1.641770],accel_mss,speed_ms,0,blend_radius_m)
    movel([0.069560, -1.349198, -2.592193, -0.770998, 1.570796, 1.640356],accel_mss,speed_ms,0,blend_radius_m)
    movel([0.068144, -1.351097, -2.590934, -0.770358, 1.570796, 1.638941],accel_mss,speed_ms,0,blend_radius_m)
    movel([0.066928, -1.352699, -2.589867, -0.769822, 1.570796, 1.637725],accel_mss,speed_ms,0,blend_radius_m)
    movel([0.065852, -1.354104, -2.588929, -0.769356, 1.570796, 1.636649],accel_mss,speed_ms,0,blend_radius_m)
    speed_ms = 0.003
    movel([0.065746, -1.357545, -2.590406, -0.764438, 1.570796, 1.636542],accel_mss,speed_ms,0,blend_radius_m)
    speed_ms = 0.007
    movel([0.065772, -1.357073, -2.590723, -0.764593, 1.570796, 1.636568],accel_mss,speed_ms,0,blend_radius_m)
    movel([0.066112, -1.356228, -2.591290, -0.764871, 1.570796, 1.636908],accel_mss,speed_ms,0,blend_radius_m)
    movel([0.067083, -1.353989, -2.592787, -0.765613, 1.570796, 1.637880],accel_mss,speed_ms,0,blend_radius_m)
    movel([0.067719, -1.352512, -2.593772, -0.766106, 1.570796, 1.638515],accel_mss,speed_ms,0,blend_radius_m)
    movel([0.068073, -1.351635, -2.594354, -0.766400, 1.570796, 1.638869],accel_mss,speed_ms,0,blend_radius_m)
    movel([0.068273, -1.351064, -2.594733, -0.766592, 1.570796, 1.639069],accel_mss,speed_ms,0,blend_radius_m)
    movel([0.068106, -1.350891, -2.594848, -0.766650, 1.570796, 1.638903],accel_mss,speed_ms,0,blend_radius_m)
    movel([0.067773, -1.350957, -2.594804, -0.766628, 1.570796, 1.638570],accel_mss,speed_ms,0,blend_radius_m)
    movel([0.067262, -1.351096, -2.594712, -0.766581, 1.570796, 1.638058],accel_mss,speed_ms,0,blend_radius_m)
    movel([0.066457, -1.351350, -2.594543, -0.766496, 1.570796, 1.637253],accel_mss,speed_ms,0,blend_radius_m)
    movel([0.065785, -1.351558, -2.594405, -0.766426, 1.570796, 1.636581],accel_mss,speed_ms,0,blend_radius_m)
    movel([0.065232, -1.351714, -2.594302, -0.766373, 1.570796, 1.636028],accel_mss,speed_ms,0,blend_radius_m)
    movel([0.064791, -1.351824, -2.594229, -0.766336, 1.570796, 1.635588],accel_mss,speed_ms,0,blend_radius_m)
    movel([0.064973, -1.350866, -2.594864, -0.766659, 1.570796, 1.635770],accel_mss,speed_ms,0,blend_radius_m)
    movel([0.065442, -1.349724, -2.595620, -0.767045, 1.570796, 1.636238],accel_mss,speed_ms,0,blend_radius_m)
    movel([0.066182, -1.348016, -2.596747, -0.767625, 1.570796, 1.636979],accel_mss,speed_ms,0,blend_radius_m)
    movel([0.066820, -1.346569, -2.597700, -0.768121, 1.570796, 1.637617],accel_mss,speed_ms,0,blend_radius_m)
    movel([0.067378, -1.345321, -2.598518, -0.768550, 1.570796, 1.638175],accel_mss,speed_ms,0,blend_radius_m)
    movel([0.067871, -1.344228, -2.599233, -0.768927, 1.570796, 1.638668],accel_mss,speed_ms,0,blend_radius_m)
    movel([0.068273, -1.343841, -2.599486, -0.769062, 1.570796, 1.639070],accel_mss,speed_ms,0,blend_radius_m)
    movel([0.070568, -1.343090, -2.599976, -0.769323, 1.570796, 1.641364],accel_mss,speed_ms,0,blend_radius_m)
    movel([0.072875, -1.342363, -2.600450, -0.769576, 1.570796, 1.643671],accel_mss,speed_ms,0,blend_radius_m)
    movel([0.073115, -1.342434, -2.600404, -0.769551, 1.570796, 1.643911],accel_mss,speed_ms,0,blend_radius_m)
    movel([0.072689, -1.343318, -2.599828, -0.769243, 1.570796, 1.643486],accel_mss,speed_ms,0,blend_radius_m)
    movel([0.072189, -1.344216, -2.599241, -0.768932, 1.570796, 1.642986],accel_mss,speed_ms,0,blend_radius_m)
    movel([0.071589, -1.345251, -2.598564, -0.768574, 1.570796, 1.642385],accel_mss,speed_ms,0,blend_radius_m)
    movel([0.070780, -1.346641, -2.597652, -0.768096, 1.570796, 1.641576],accel_mss,speed_ms,0,blend_radius_m)
    movel([0.070360, -1.347409, -2.597148, -0.767833, 1.570796, 1.641156],accel_mss,speed_ms,0,blend_radius_m)
